// TIA Portal V16 program export: 1 tag tables, 0 data types, 4 data blocks, 6 code blocks (in call order from the OBs), 8 instance data blocks

VAR_GLOBAL   // PLC tag table "Default tag table"
   System_Byte AT %MB1 : Byte;
   FirstScan AT %M1.0 : Bool;
   DiagStatusUpdate AT %M1.1 : Bool;
   AlwaysTRUE AT %M1.2 : Bool;
   AlwaysFALSE AT %M1.3 : Bool;
   Clock_Byte AT %MB0 : Byte;
   Clock_10Hz AT %M0.0 : Bool;
   Clock_5Hz AT %M0.1 : Bool;
   "Clock_2.5Hz" AT %M0.2 : Bool;
   Clock_2Hz AT %M0.3 : Bool;
   "Clock_1.25Hz" AT %M0.4 : Bool;
   Clock_1Hz AT %M0.5 : Bool;
   "Clock_0.625Hz" AT %M0.6 : Bool;
   "Clock_0.5Hz" AT %M0.7 : Bool;
   Aux_1 AT %M2.0 : Bool;
   START_COMM AT %M2.1 : Bool;
   BS_03 AT %M2.6 : Bool;
   Comm_ok AT %M2.3 : Bool;
   Count_Modbus AT %MW50 : Word;
   RST_Count AT %M49.0 : Bool;
   Tag_2 AT %M49.1 : Bool;
   Tag_3 AT %M49.2 : Bool;
   Tag_4 AT %M49.3 : Bool;
   Tag_5 AT %M49.4 : Bool;
   MB_DONE_COUNT AT %MW54 : Word;
   Tag_7 AT %M49.7 : Bool;
   MB_ERROR_COUNT AT %MW58 : Word;
   MB_STATUS AT %MW62 : Word;
   Tag_10 AT %M30.0 : Bool;
   Tag_11 AT %MW70 : Word;
   Tag_12 AT %MW74 : Word;
   Tag_13 AT %MW78 : Word;
   Liga_01 AT %M3.0 : Bool;
   Desliga_01 AT %M3.1 : Bool;
   Liga_02 AT %M3.2 : Bool;
   Desliga_02 AT %M3.3 : Bool;
   Liga_03 AT %M3.4 : Bool;
   Desliga_03 AT %M3.5 : Bool;
   Liga_04 AT %M3.6 : Bool;
   Desliga_04 AT %M3.7 : Bool;
   Liga_05 AT %M4.0 : Bool;
   Desliga_05 AT %M4.1 : Bool;
   Liga_06 AT %M4.2 : Bool;
   Desliga_06 AT %M4.3 : Bool;
   Liga_07 AT %M4.4 : Bool;
   Desliga_07 AT %M4.5 : Bool;
   Liga_08 AT %M4.6 : Bool;
   Desliga_08 AT %M4.7 : Bool;
   Liga_09 AT %M5.0 : Bool;
   Desliga_09 AT %M5.1 : Bool;
   Liga_10 AT %M5.2 : Bool;
   Desliga_10 AT %M5.3 : Bool;
   Liga_11 AT %M5.4 : Bool;
   Desliga_11 AT %M5.5 : Bool;
   Liga_12 AT %M5.6 : Bool;
   Desliga_12 AT %M5.7 : Bool;
   Liga_13 AT %M6.0 : Bool;
   Desliga_13 AT %M6.1 : Bool;
   Liga_14 AT %M6.2 : Bool;
   Desliga_14 AT %M6.3 : Bool;
   Oper_Mode_01 AT %MW80 : Word;
   SP_01 AT %MW82 : Word;
   Oper_Mode_02 AT %MW84 : Word;
   SP_02 AT %MW86 : Word;
   Oper_Mode_03 AT %MW88 : Word;
   SP_03 AT %MW90 : Word;
   Oper_Mode_04 AT %MW92 : Word;
   SP_04 AT %MW94 : Word;
   Oper_Mode_05 AT %MW96 : Word;
   SP_05 AT %MW98 : Word;
   Oper_Mode_06 AT %MW100 : Word;
   SP_06 AT %MW102 : Word;
   Oper_Mode_07 AT %MW104 : Word;
   SP_07 AT %MW106 : Word;
   Oper_Mode_08 AT %MW108 : Word;
   SP_08 AT %MW110 : Word;
   Oper_Mode_09 AT %MW112 : Word;
   SP_09 AT %MW114 : Word;
   Oper_Mode_10 AT %MW116 : Word;
   SP_10 AT %MW118 : Word;
   Oper_Mode_11 AT %MW120 : Word;
   SP_11 AT %MW122 : Word;
   Oper_Mode_12 AT %MW124 : Word;
   SP_12 AT %MW126 : Word;
   Oper_Mode_13 AT %MW128 : Word;
   SP_13 AT %MW130 : Word;
   Oper_Mode_14 AT %MW132 : Word;
   SP_14 AT %MW134 : Word;
   Tag_1 AT %M7.1 : Bool;
   Timeout_Desligado_Counter AT %M6.4 : Bool;
   Timeout_Ligado_Counter AT %M6.5 : Bool;
   Tag_8 AT %M6.6 : Bool;
   Tag_6 AT %M6.7 : Bool;
   MB_CT_DONE AT %M7.2 : Bool;
   MB_CT_ERROR AT %M7.3 : Bool;
   Sts_Auto AT %M7.4 : Bool;
   Tag_9 AT %MW240 : Word;
   Tag_14 AT %MD242 : Real;
   "1" AT %MD246 : Real;
   Tag_15 AT %MW242 : Word;
END_VAR

DATA_BLOCK "Data_block_1"   // DB1
{ S7_Optimized_Access := 'FALSE' }
VERSION : 0.1
// stored: AutoNumber true, DBAccessibleFromOPCUA true, IsOnlyStoredInLoadMemory false, IsWriteProtectedInAS false
   VAR RETAIN
      Descritivo_TBR : Array[0..13] of String;
      Descritivo_TOP : Array[0..1] of String;
   END_VAR
BEGIN
END_DATA_BLOCK

DATA_BLOCK "Modbus"   // DB5
{ S7_Optimized_Access := 'TRUE' }
VERSION : 0.1
// stored: AutoNumber true, DBAccessibleFromOPCUA true, IsOnlyStoredInLoadMemory false, IsRetainMemResEnabled false, IsWriteProtectedInAS false, MemoryReserve 100
   VAR
      Done : Bool;
      Busy : Bool;
      Error : Bool;
      Status : Word;
      Input_Reading : Struct
         "30000" : Array[0..149] of Word;
      END_STRUCT;
   END_VAR
BEGIN
END_DATA_BLOCK

DATA_BLOCK "Modbus_Send_Receive"   // DB10
{ S7_Optimized_Access := 'FALSE' }
VERSION : 0.1
// stored: AutoNumber true, DBAccessibleFromOPCUA true, IsOnlyStoredInLoadMemory false, IsWriteProtectedInAS false
   VAR
      "30001" : Word;
      "30002" : Word;   // COMM_OK = 3FFF
      "32001" : Word;   // STS_UNIT_01
      "32002" : Word;   // OPER_UNIT_01
      "32003" : Word;   // SP_UNIT_01
      "32004" : Word;   // ERROR_UNIT_01
      "32005" : Word;   // PV_UNIT_01
      "32006" : Word;   // SERROR_UNIT_01
      "32007" : Word;   // STS_UNIT_02
      "32008" : Word;   // OPER_UNIT_02
      "32009" : Word;   // SP_UNIT_02
      "32010" : Word;   // ERROR_UNIT_02
      "32011" : Word;   // PV_UNIT_02
      "32012" : Word;   // SERROR_UNIT_02
      "32013" : Word;
      "32014" : Word;
      "32015" : Word;
      "32016" : Word;
      "32017" : Word;
      "32018" : Word;
      "32019" : Word;
      "32020" : Word;
      "32021" : Word;
      "32022" : Word;
      "32023" : Word;
      "32024" : Word;
      "32025" : Word;
      "32026" : Word;
      "32027" : Word;
      "32028" : Word;
      "32029" : Word;
      "32030" : Word;
      "32031" : Word;
      "32032" : Word;
      "32033" : Word;
      "32034" : Word;
      "32035" : Word;
      "32036" : Word;
      "32037" : Word;
      "32038" : Word;
      "32039" : Word;
      "32040" : Word;
      "32041" : Word;
      "32042" : Word;
      "32043" : Word;
      "32044" : Word;
      "32045" : Word;
      "32046" : Word;
      "32047" : Word;
      "32048" : Word;
      "32049" : Word;
      "32050" : Word;
      "32051" : Word;
      "32052" : Word;
      "32053" : Word;
      "32054" : Word;
      "32055" : Word;
      "32056" : Word;
      "32057" : Word;
      "32058" : Word;
      "32059" : Word;
      "32060" : Word;
      "32061" : Word;
      "32062" : Word;
      "32063" : Word;
      "32064" : Word;
      "32065" : Word;
      "32066" : Word;
      "32067" : Word;
      "32068" : Word;
      "32069" : Word;
      "32070" : Word;
      "32071" : Word;
      "32072" : Word;
      "32073" : Word;
      "32074" : Word;
      "32075" : Word;
      "32076" : Word;
      "32077" : Word;
      "32078" : Word;
      "32079" : Word;
      "32080" : Word;
      "32081" : Word;
      "32082" : Word;
      "32083" : Word;
      "32084" : Word;
      "40001" : Word;   // COMM
      "42001" : Word;   // STS
      "42002" : Word;   // OPER_MODE
      "42003" : Word;   // SP
      "42004" : Word;   // STS
      "42005" : Word;   // OPER_MODE
      "42006" : Word;   // SP
      "42007" : Word;   // STS
      "42008" : Word;   // OPER_MODE
      "42009" : Word;   // SP
      "42010" : Word;   // STS
      "42011" : Word;   // OPER_MODE
      "42012" : Word;   // SP
      "42013" : Word;   // STS
      "42014" : Word;   // OPER_MODE
      "42015" : Word;   // SP
      "42016" : Word;   // STS
      "42017" : Word;   // OPER_MODE
      "42018" : Word;   // SP
      "42019" : Word;   // STS
      "42020" : Word;   // OPER_MODE
      "42021" : Word;   // SP
      "42022" : Word;   // STS
      "42023" : Word;   // OPER_MODE
      "42024" : Word;   // SP
      "42025" : Word;   // STS
      "42026" : Word;   // OPER_MODE
      "42027" : Word;   // SP
      "42028" : Word;   // STS
      "42029" : Word;   // OPER_MODE
      "42030" : Word;   // SP
      "42031" : Word;   // STS
      "42032" : Word;   // OPER_MODE
      "42033" : Word;   // SP
      "42034" : Word;   // STS
      "42035" : Word;   // OPER_MODE
      "42036" : Word;   // SP
      "42037" : Word;   // STS
      "42038" : Word;   // OPER_MODE
      "42039" : Word;   // SP
      "42040" : Word;   // STS
      "42041" : Word;   // OPER_MODE
      "42042" : Word;   // SP
      Extrusora_1 : Struct
         Ligado : Bool;
         Fan : Bool;
         Heating : Bool;
         Cooling : Bool;
         Sts_Fan : Bool;
         Sts_Heating : Bool;
         Sts_Cooling : Bool;
         Slave : Bool;
         Master : Bool;
         SP : Real;
         PV : Real;
      END_STRUCT;
      Extrusora_2 : Struct
         Ligado : Bool;
         Fan : Bool;
         Heating : Bool;
         Cooling : Bool;
         Sts_Fan : Bool;
         Sts_Heating : Bool;
         Sts_Cooling : Bool;
         Slave : Bool;
         Master : Bool;
         SP : Real;
         PV : Real;
      END_STRUCT;
      Extrusora_3 : Struct
         Ligado : Bool;
         Fan : Bool;
         Heating : Bool;
         Cooling : Bool;
         Sts_Fan : Bool;
         Sts_Heating : Bool;
         Sts_Cooling : Bool;
         Slave : Bool;
         Master : Bool;
         SP : Real;
         PV : Real;
      END_STRUCT;
      Extrusora_4 : Struct
         Ligado : Bool;
         Fan : Bool;
         Heating : Bool;
         Cooling : Bool;
         Sts_Fan : Bool;
         Sts_Heating : Bool;
         Sts_Cooling : Bool;
         Slave : Bool;
         Master : Bool;
         SP : Real;
         PV : Real;
      END_STRUCT;
      Extrusora_5 : Struct
         Ligado : Bool;
         Fan : Bool;
         Heating : Bool;
         Cooling : Bool;
         Sts_Fan : Bool;
         Sts_Heating : Bool;
         Sts_Cooling : Bool;
         Slave : Bool;
         Master : Bool;
         SP : Real;
         PV : Real;
      END_STRUCT;
      Extrusora_6 : Struct
         Ligado : Bool;
         Fan : Bool;
         Heating : Bool;
         Cooling : Bool;
         Sts_Fan : Bool;
         Sts_Heating : Bool;
         Sts_Cooling : Bool;
         Slave : Bool;
         Master : Bool;
         SP : Real;
         PV : Real;
      END_STRUCT;
      Extrusora_7 : Struct
         Ligado : Bool;
         Fan : Bool;
         Heating : Bool;
         Cooling : Bool;
         Sts_Fan : Bool;
         Sts_Heating : Bool;
         Sts_Cooling : Bool;
         Slave : Bool;
         Master : Bool;
         SP : Real;
         PV : Real;
      END_STRUCT;
      Extrusora_8 : Struct
         Ligado : Bool;
         Fan : Bool;
         Heating : Bool;
         Cooling : Bool;
         Sts_Fan : Bool;
         Sts_Heating : Bool;
         Sts_Cooling : Bool;
         Slave : Bool;
         Master : Bool;
         SP : Real;
         PV : Real;
      END_STRUCT;
      Extrusora_9 : Struct
         Ligado : Bool;
         Fan : Bool;
         Heating : Bool;
         Cooling : Bool;
         Sts_Fan : Bool;
         Sts_Heating : Bool;
         Sts_Cooling : Bool;
         Slave : Bool;
         Master : Bool;
         SP : Real;
         PV : Real;
      END_STRUCT;
      Extrusora_10 : Struct
         Ligado : Bool;
         Fan : Bool;
         Heating : Bool;
         Cooling : Bool;
         Sts_Fan : Bool;
         Sts_Heating : Bool;
         Sts_Cooling : Bool;
         Slave : Bool;
         Master : Bool;
         SP : Real;
         PV : Real;
      END_STRUCT;
      Extrusora_11 : Struct
         Ligado : Bool;
         Fan : Bool;
         Heating : Bool;
         Cooling : Bool;
         Sts_Fan : Bool;
         Sts_Heating : Bool;
         Sts_Cooling : Bool;
         Slave : Bool;
         Master : Bool;
         SP : Real;
         PV : Real;
      END_STRUCT;
      Extrusora_12 : Struct
         Ligado : Bool;
         Fan : Bool;
         Heating : Bool;
         Cooling : Bool;
         Sts_Fan : Bool;
         Sts_Heating : Bool;
         Sts_Cooling : Bool;
         Slave : Bool;
         Master : Bool;
         SP : Real;
         PV : Real;
      END_STRUCT;
      Extrusora_13 : Struct
         Ligado : Bool;
         Fan : Bool;
         Heating : Bool;
         Cooling : Bool;
         Sts_Fan : Bool;
         Sts_Heating : Bool;
         Sts_Cooling : Bool;
         Slave : Bool;
         Master : Bool;
         SP : Real;
         PV : Real;
      END_STRUCT;
      Extrusora_14 : Struct
         Ligado : Bool;
         Fan : Bool;
         Heating : Bool;
         Cooling : Bool;
         Sts_Fan : Bool;
         Sts_Heating : Bool;
         Sts_Cooling : Bool;
         Slave : Bool;
         Master : Bool;
         SP : Real;
         PV : Real;
      END_STRUCT;
      Malfunction_1 : Bool;
      Malfunction_2 : Bool;
      Malfunction_3 : Bool;
      Malfunction_4 : Bool;
      Malfunction_5 : Bool;
      Malfunction_6 : Bool;
      Malfunction_7 : Bool;
      Malfunction_8 : Bool;
      Malfunction_9 : Bool;
      Malfunction_10 : Bool;
      Malfunction_11 : Bool;
      Malfunction_12 : Bool;
      Malfunction_13 : Bool;
      Malfunction_14 : Bool;
   END_VAR
BEGIN
END_DATA_BLOCK

DATA_BLOCK "Modbus_Send_Receive_1"   // DB13
{ S7_Optimized_Access := 'FALSE' }
VERSION : 0.1
// stored: AutoNumber false, DBAccessibleFromOPCUA true, IsOnlyStoredInLoadMemory false, IsWriteProtectedInAS false
   VAR
      Reading_Struct : Struct
         "32001" : Word;   // STS_UNIT_01
         "32002" : Word;   // OPER_UNIT_01
         "32003" : Word;   // SP_UNIT_01
         "32004" : Word;   // ERROR_UNIT_01
         "32005" : Word;   // PV_UNIT_01
         "32006" : Word;   // SERROR_UNIT_01
         "32007" : Word;   // STS_UNIT_02
         "32008" : Word;   // OPER_UNIT_02
         "32009" : Word;   // SP_UNIT_02
         "32010" : Word;   // ERROR_UNIT_02
         "32011" : Word;   // PV_UNIT_02
         "32012" : Word;   // SERROR_UNIT_02
         "32013" : Word;   // STS_UNIT_01
         "32014" : Word;   // OPER_UNIT_01
         "32015" : Word;   // SP_UNIT_01
         "32016" : Word;   // ERROR_UNIT_01
         "32017" : Word;   // PV_UNIT_01
         "32018" : Word;   // SERROR_UNIT_01
         "32019" : Word;   // STS_UNIT_02
         "32020" : Word;   // OPER_UNIT_02
         "32021" : Word;   // SP_UNIT_02
         "32022" : Word;   // ERROR_UNIT_02
         "32023" : Word;   // PV_UNIT_02
         "32024" : Word;   // SERROR_UNIT_02
         "32025" : Word;   // STS_UNIT_01
         "32026" : Word;   // OPER_UNIT_01
         "32027" : Word;   // SP_UNIT_01
         "32028" : Word;   // ERROR_UNIT_01
         "32029" : Word;   // PV_UNIT_01
         "32030" : Word;   // SERROR_UNIT_01
         "32031" : Word;   // STS_UNIT_02
         "32032" : Word;   // OPER_UNIT_02
         "32033" : Word;   // SP_UNIT_02
         "32034" : Word;   // ERROR_UNIT_02
         "32035" : Word;   // PV_UNIT_02
         "32036" : Word;   // SERROR_UNIT_02
         "32037" : Word;   // STS_UNIT_01
         "32038" : Word;   // OPER_UNIT_01
         "32039" : Word;   // SP_UNIT_01
         "32040" : Word;   // ERROR_UNIT_01
         "32041" : Word;   // PV_UNIT_01
         "32042" : Word;   // SERROR_UNIT_01
         "32043" : Word;   // STS_UNIT_02
         "32044" : Word;   // OPER_UNIT_02
         "32045" : Word;   // SP_UNIT_02
         "32046" : Word;   // ERROR_UNIT_02
         "32047" : Word;   // PV_UNIT_02
         "32048" : Word;   // SERROR_UNIT_02
         "32049" : Word;   // STS_UNIT_01
         "32050" : Word;   // OPER_UNIT_01
         "32051" : Word;   // SP_UNIT_01
         "32052" : Word;   // ERROR_UNIT_01
         "32053" : Word;   // PV_UNIT_01
         "32054" : Word;   // SERROR_UNIT_01
         "32055" : Word;   // STS_UNIT_02
         "32056" : Word;   // OPER_UNIT_02
         "32057" : Word;   // SP_UNIT_02
         "32058" : Word;   // ERROR_UNIT_02
         "32059" : Word;   // PV_UNIT_02
         "32060" : Word;   // SERROR_UNIT_02
         "32061" : Word;   // STS_UNIT_01
         "32062" : Word;   // OPER_UNIT_01
         "32063" : Word;   // SP_UNIT_01
         "32064" : Word;   // ERROR_UNIT_01
         "32065" : Word;   // PV_UNIT_01
         "32066" : Word;   // SERROR_UNIT_01
         "32067" : Word;   // STS_UNIT_02
         "32068" : Word;   // OPER_UNIT_02
         "32069" : Word;   // SP_UNIT_02
         "32070" : Word;   // ERROR_UNIT_02
         "32071" : Word;   // PV_UNIT_02
         "32072" : Word;   // SERROR_UNIT_02
         "32073" : Word;   // STS_UNIT_01
         "32074" : Word;   // OPER_UNIT_01
         "32075" : Word;   // SP_UNIT_01
         "32076" : Word;   // ERROR_UNIT_01
         "32077" : Word;   // PV_UNIT_01
         "32078" : Word;   // SERROR_UNIT_01
         "32079" : Word;   // STS_UNIT_02
         "32080" : Word;   // OPER_UNIT_02
         "32081" : Word;   // SP_UNIT_02
         "32082" : Word;   // ERROR_UNIT_02
         "32083" : Word;   // PV_UNIT_02
         "32084" : Word;   // SERROR_UNIT_02
         "40001" : Word;
         "42001" : Word;   // STS
         "42002" : Word;   // OPER_MODE
         "42003" : Word;   // SP
         "42004" : Word;
         "42005" : Word;
         "42006" : Word;
         "42007" : Word;
         "42008" : Word;
         "42009" : Word;
         "42010" : Word;
         "42011" : Word;
         "42012" : Word;
         "42013" : Word;
         "42014" : Word;
         "42015" : Word;
         "42016" : Word;
         "42017" : Word;
         "42018" : Word;
         "42019" : Word;
         "42020" : Word;
         "42021" : Word;
         "42022" : Word;
         "42023" : Word;
         "42024" : Word;
         "42025" : Word;
         "42026" : Word;
         "42027" : Word;
         "42028" : Word;
         "42029" : Word;
         "42030" : Word;
         "42031" : Word;
         "42032" : Word;
         "42033" : Word;
         "42034" : Word;
         "42035" : Word;
         "42036" : Word;
         "42037" : Word;
         "42038" : Word;
         "42039" : Word;
         "42040" : Word;
         "42041" : Word;
         "42042" : Word;
      END_STRUCT;
      Reading_Struct_2 : Struct
         "30001" : Word;
         "30002" : Word;   // COMM_OK = 3FFF
      END_STRUCT;
      Extrusora_1 : Struct
         Ligado : Bool;
         Fan : Bool;
         Heating : Bool;
         Cooling : Bool;
         Sts_Fan : Bool;
         Sts_Heating : Bool;
         Sts_Cooling : Bool;
         Slave : Bool;
         Master : Bool;
         SP : Word;
         PV : Word;
      END_STRUCT;
      Extrusora_2 : Struct
         Ligado : Bool;
         Fan : Bool;
         Heating : Bool;
         Cooling : Bool;
         Sts_Fan : Bool;
         Sts_Heating : Bool;
         Sts_Cooling : Bool;
         Slave : Bool;
         Master : Bool;
         SP : Word;
         PV : Word;
      END_STRUCT;
      Extrusora_3 : Struct
         Ligado : Bool;
         Fan : Bool;
         Heating : Bool;
         Cooling : Bool;
         Sts_Fan : Bool;
         Sts_Heating : Bool;
         Sts_Cooling : Bool;
         Slave : Bool;
         Master : Bool;
         SP : Word;
         PV : Word;
      END_STRUCT;
      Extrusora_4 : Struct
         Ligado : Bool;
         Fan : Bool;
         Heating : Bool;
         Cooling : Bool;
         Sts_Fan : Bool;
         Sts_Heating : Bool;
         Sts_Cooling : Bool;
         Slave : Bool;
         Master : Bool;
         SP : Word;
         PV : Word;
      END_STRUCT;
      Extrusora_5 : Struct
         Ligado : Bool;
         Fan : Bool;
         Heating : Bool;
         Cooling : Bool;
         Sts_Fan : Bool;
         Sts_Heating : Bool;
         Sts_Cooling : Bool;
         Slave : Bool;
         Master : Bool;
         SP : Word;
         PV : Word;
      END_STRUCT;
      Extrusora_6 : Struct
         Ligado : Bool;
         Fan : Bool;
         Heating : Bool;
         Cooling : Bool;
         Sts_Fan : Bool;
         Sts_Heating : Bool;
         Sts_Cooling : Bool;
         Slave : Bool;
         Master : Bool;
         SP : Word;
         PV : Word;
      END_STRUCT;
      Extrusora_7 : Struct
         Ligado : Bool;
         Fan : Bool;
         Heating : Bool;
         Cooling : Bool;
         Sts_Fan : Bool;
         Sts_Heating : Bool;
         Sts_Cooling : Bool;
         Slave : Bool;
         Master : Bool;
         SP : Word;
         PV : Word;
      END_STRUCT;
      Extrusora_8 : Struct
         Ligado : Bool;
         Fan : Bool;
         Heating : Bool;
         Cooling : Bool;
         Sts_Fan : Bool;
         Sts_Heating : Bool;
         Sts_Cooling : Bool;
         Slave : Bool;
         Master : Bool;
         SP : Word;
         PV : Word;
      END_STRUCT;
      Extrusora_9 : Struct
         Ligado : Bool;
         Fan : Bool;
         Heating : Bool;
         Cooling : Bool;
         Sts_Fan : Bool;
         Sts_Heating : Bool;
         Sts_Cooling : Bool;
         Slave : Bool;
         Master : Bool;
         SP : Word;
         PV : Word;
      END_STRUCT;
      Extrusora_10 : Struct
         Ligado : Bool;
         Fan : Bool;
         Heating : Bool;
         Cooling : Bool;
         Sts_Fan : Bool;
         Sts_Heating : Bool;
         Sts_Cooling : Bool;
         Slave : Bool;
         Master : Bool;
         SP : Word;
         PV : Word;
      END_STRUCT;
      Extrusora_11 : Struct
         Ligado : Bool;
         Fan : Bool;
         Heating : Bool;
         Cooling : Bool;
         Sts_Fan : Bool;
         Sts_Heating : Bool;
         Sts_Cooling : Bool;
         Slave : Bool;
         Master : Bool;
         SP : Word;
         PV : Word;
      END_STRUCT;
      Extrusora_12 : Struct
         Ligado : Bool;
         Fan : Bool;
         Heating : Bool;
         Cooling : Bool;
         Sts_Fan : Bool;
         Sts_Heating : Bool;
         Sts_Cooling : Bool;
         Slave : Bool;
         Master : Bool;
         SP : Word;
         PV : Word;
      END_STRUCT;
      Extrusora_13 : Struct
         Ligado : Bool;
         Fan : Bool;
         Heating : Bool;
         Cooling : Bool;
         Sts_Fan : Bool;
         Sts_Heating : Bool;
         Sts_Cooling : Bool;
         Slave : Bool;
         Master : Bool;
         SP : Word;
         PV : Word;
      END_STRUCT;
      Extrusora_14 : Struct
         Ligado : Bool;
         Fan : Bool;
         Heating : Bool;
         Cooling : Bool;
         Sts_Fan : Bool;
         Sts_Heating : Bool;
         Sts_Cooling : Bool;
         Slave : Bool;
         Master : Bool;
         SP : Word;
         PV : Word;
      END_STRUCT;
      Malfunction_1 : Bool;
      Malfunction_2 : Bool;
      Malfunction_3 : Bool;
      Malfunction_4 : Bool;
      Malfunction_5 : Bool;
      Malfunction_6 : Bool;
      Malfunction_7 : Bool;
      Malfunction_8 : Bool;
      Malfunction_9 : Bool;
      Malfunction_10 : Bool;
      Malfunction_11 : Bool;
      Malfunction_12 : Bool;
      Malfunction_13 : Bool;
      Malfunction_14 : Bool;
   END_VAR
BEGIN
END_DATA_BLOCK

ORGANIZATION_BLOCK "Main"   // OB1, LAD, ProgramCycle
TITLE = "Main Program Sweep (Cycle)"
{ S7_Optimized_Access := 'TRUE' }
VERSION : 0.1
// stored: AutoNumber true, IsIECCheckEnabled false, SetENOAutomatically false
BEGIN

REGION Network 1: Start modbus comm
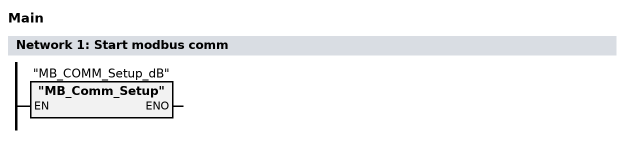
   RUNG wire#powerrail
      "MB_COMM_Setup_dB"()
   END_RUNG
   // the same network as SCL:
   "MB_COMM_Setup_dB"();   // "MB_Comm_Setup"
END_REGION
END_ORGANIZATION_BLOCK

FUNCTION_BLOCK "MB_Comm_Setup"   // FB1, LAD
{ S7_Optimized_Access := 'FALSE' }
VERSION : 0.1
// stored: AutoNumber true, IsIECCheckEnabled false, SetENOAutomatically false, UDAEnableTagReadback false
   VAR DB_SPECIFIC
      Input_Registers_3000X_In { ExternalAccessible := 'False'; ExternalVisible := 'False'; ExternalWritable := 'False'} : Struct
         "3000X" { ExternalAccessible := 'False'; ExternalVisible := 'False'; ExternalWritable := 'False'} : Array[0..150] of Word;
      END_STRUCT;
   END_VAR
   VAR
      Input_Registers_In_AT AT Input_Registers_3000X_In : Struct
         "30001" : Array[0..15] of Bool;
         "30001_2" : Array[0..15] of Bool;   // Status of the Adaptor
         "30002" : Array[0..15] of Bool;   // Indoor Unit Connection Status
         "30003" : Array[0..15] of Bool;   // Empty
         "30004" : Array[0..15] of Bool;   // Empty
         "30005" : Array[0..15] of Bool;   // Empty
         "30006" : Array[0..15] of Bool;   // Indoor Unit Communication Status
         "31001" : Array[0..15] of Bool;   // Various
         "31002" : Array[0..15] of Bool;   // 1st word - Indoor unit cooling setpoint upper limit, 2 - word indoor unit cooling setpoint lower limit
         "31003" : Array[0..15] of Bool;   // 1st word - Indoor unit heating setpoint upper limit, 2 - word indoor unit heating setpoint lower limit
         "31004" : Array[0..15] of Bool;   // Various
         "31005" : Array[0..15] of Bool;   // 1st word - Indoor unit cooling setpoint upper limit, 2 - word indoor unit cooling setpoint lower limit
         "31006" : Array[0..15] of Bool;   // 1st word - Indoor unit heating setpoint upper limit, 2 - word indoor unit heating setpoint lower limit
         "31007" : Array[0..15] of Bool;   // Various
         "31008" : Array[0..15] of Bool;   // 1st word - Indoor unit cooling setpoint upper limit, 2 - word indoor unit cooling setpoint lower limit
         "31009" : Array[0..15] of Bool;   // 1st word - Indoor unit heating setpoint upper limit, 2 - word indoor unit heating setpoint lower limit
         "31010" : Array[0..15] of Bool;   // Various
         "31011" : Array[0..15] of Bool;   // 1st word - Indoor unit cooling setpoint upper limit, 2 - word indoor unit cooling setpoint lower limit
         "31012" : Array[0..15] of Bool;   // 1st word - Indoor unit heating setpoint upper limit, 2 - word indoor unit heating setpoint lower limit
         "31013" : Array[0..15] of Bool;   // Various
         "31014" : Array[0..15] of Bool;   // 1st word - Indoor unit cooling setpoint upper limit, 2 - word indoor unit cooling setpoint lower limit
         "31015" : Array[0..15] of Bool;   // 1st word - Indoor unit heating setpoint upper limit, 2 - word indoor unit heating setpoint lower limit
         "31016" : Array[0..15] of Bool;   // Various
         "31017" : Array[0..15] of Bool;   // 1st word - Indoor unit cooling setpoint upper limit, 2 - word indoor unit cooling setpoint lower limit
         "31018" : Array[0..15] of Bool;   // 1st word - Indoor unit heating setpoint upper limit, 2 - word indoor unit heating setpoint lower limit
         "31019" : Array[0..15] of Bool;   // Various
         "31020" : Array[0..15] of Bool;   // 1st word - Indoor unit cooling setpoint upper limit, 2 - word indoor unit cooling setpoint lower limit
         "31021" : Array[0..15] of Bool;   // 1st word - Indoor unit heating setpoint upper limit, 2 - word indoor unit heating setpoint lower limit
         "31022" : Array[0..15] of Bool;   // Various
         "31023" : Array[0..15] of Bool;   // 1st word - Indoor unit cooling setpoint upper limit, 2 - word indoor unit cooling setpoint lower limit
         "31024" : Array[0..15] of Bool;   // 1st word - Indoor unit heating setpoint upper limit, 2 - word indoor unit heating setpoint lower limit
         "31025" : Array[0..15] of Bool;   // Various
         "31026" : Array[0..15] of Bool;   // 1st word - Indoor unit cooling setpoint upper limit, 2 - word indoor unit cooling setpoint lower limit
         "31027" : Array[0..15] of Bool;   // 1st word - Indoor unit heating setpoint upper limit, 2 - word indoor unit heating setpoint lower limit
         "31028" : Array[0..15] of Bool;   // Various
         "31029" : Array[0..15] of Bool;   // 1st word - Indoor unit cooling setpoint upper limit, 2 - word indoor unit cooling setpoint lower limit
         "31030" : Array[0..15] of Bool;   // 1st word - Indoor unit heating setpoint upper limit, 2 - word indoor unit heating setpoint lower limit
         "31031" : Array[0..15] of Bool;   // Various
         "31032" : Array[0..15] of Bool;   // 1st word - Indoor unit cooling setpoint upper limit, 2 - word indoor unit cooling setpoint lower limit
         "31033" : Array[0..15] of Bool;   // 1st word - Indoor unit heating setpoint upper limit, 2 - word indoor unit heating setpoint lower limit
         "31034" : Array[0..15] of Bool;   // Various
         "31035" : Array[0..15] of Bool;   // 1st word - Indoor unit cooling setpoint upper limit, 2 - word indoor unit cooling setpoint lower limit
         "31036" : Array[0..15] of Bool;   // 1st word - Indoor unit heating setpoint upper limit, 2 - word indoor unit heating setpoint lower limit
         "31037" : Array[0..15] of Bool;   // Various
         "31038" : Array[0..15] of Bool;   // 1st word - Indoor unit cooling setpoint upper limit, 2 - word indoor unit cooling setpoint lower limit
         "31039" : Array[0..15] of Bool;   // 1st word - Indoor unit heating setpoint upper limit, 2 - word indoor unit heating setpoint lower limit
         "31040" : Array[0..15] of Bool;   // Various
         "31041" : Array[0..15] of Bool;   // 1st word - Indoor unit cooling setpoint upper limit, 2 - word indoor unit cooling setpoint lower limit
         "31042" : Array[0..15] of Bool;   // 1st word - Indoor unit heating setpoint upper limit, 2 - word indoor unit heating setpoint lower limit
         "31043" : Array[0..15] of Bool;   // Various
         "31044" : Array[0..15] of Bool;   // 1st word - Indoor unit cooling setpoint upper limit, 2 - word indoor unit cooling setpoint lower limit
         "31045" : Array[0..15] of Bool;   // 1st word - Indoor unit heating setpoint upper limit, 2 - word indoor unit heating setpoint lower limit
         "31046" : Array[0..15] of Bool;   // Various
         "31047" : Array[0..15] of Bool;   // 1st word - Indoor unit cooling setpoint upper limit, 2 - word indoor unit cooling setpoint lower limit
         "31048" : Array[0..15] of Bool;   // 1st word - Indoor unit heating setpoint upper limit, 2 - word indoor unit heating setpoint lower limit
         "32001" : Array[0..15] of Bool;   // Important stuff
         "32002" : Array[0..15] of Bool;   // Important stuff_2
         "32003" : Array[0..15] of Bool;   // Setpoint Temperature
         "32004" : Array[0..15] of Bool;   // Important Stuff_3
         "32005" : Array[0..15] of Bool;   // Room Temperature
         "32006" : Array[0..15] of Bool;   // Error
         "32007" : Array[0..15] of Bool;   // Important stuff
         "32008" : Array[0..15] of Bool;   // Important stuff_2
         "32009" : Array[0..15] of Bool;   // Setpoint Temperature
         "32010" : Array[0..15] of Bool;   // Important Stuff_3
         "32011" : Array[0..15] of Bool;   // Room Temperature
         "32012" : Array[0..15] of Bool;   // Error
         "32013" : Array[0..15] of Bool;   // Important stuff
         "32014" : Array[0..15] of Bool;   // Important stuff_2
         "32015" : Array[0..15] of Bool;   // Setpoint Temperature
         "32016" : Array[0..15] of Bool;   // Important Stuff_3
         "32017" : Array[0..15] of Bool;   // Room Temperature
         "32018" : Array[0..15] of Bool;   // Error
         "32019" : Array[0..15] of Bool;   // Important stuff
         "32020" : Array[0..15] of Bool;   // Important stuff_2
         "32021" : Array[0..15] of Bool;   // Setpoint Temperature
         "32022" : Array[0..15] of Bool;   // Important Stuff_3
         "32023" : Array[0..15] of Bool;   // Room Temperature
         "32024" : Array[0..15] of Bool;   // Error
         "32025" : Array[0..15] of Bool;   // Important stuff
         "32026" : Array[0..15] of Bool;   // Important stuff_2
         "32027" : Array[0..15] of Bool;   // Setpoint Temperature
         "32028" : Array[0..15] of Bool;   // Important Stuff_3
         "32029" : Array[0..15] of Bool;   // Room Temperature
         "32030" : Array[0..15] of Bool;   // Error
         "32031" : Array[0..15] of Bool;   // Important stuff
         "32032" : Array[0..15] of Bool;   // Important stuff_2
         "32033" : Array[0..15] of Bool;   // Setpoint Temperature
         "32034" : Array[0..15] of Bool;   // Important Stuff_3
         "32035" : Array[0..15] of Bool;   // Room Temperature
         "32036" : Array[0..15] of Bool;   // Error
         "32037" : Array[0..15] of Bool;   // Important stuff
         "32038" : Array[0..15] of Bool;   // Important stuff_2
         "32039" : Array[0..15] of Bool;   // Setpoint Temperature
         "32040" : Array[0..15] of Bool;   // Important Stuff_3
         "32041" : Array[0..15] of Bool;   // Room Temperature
         "32042" : Array[0..15] of Bool;   // Error
         "32043" : Array[0..15] of Bool;   // Important stuff
         "32044" : Array[0..15] of Bool;   // Important stuff_2
         "32045" : Array[0..15] of Bool;   // Setpoint Temperature
         "32046" : Array[0..15] of Bool;   // Important Stuff_3
         "32047" : Array[0..15] of Bool;   // Room Temperature
         "32048" : Array[0..15] of Bool;   // Error
         "32049" : Array[0..15] of Bool;   // Important stuff
         "32050" : Array[0..15] of Bool;   // Important stuff_2
         "32051" : Array[0..15] of Bool;   // Setpoint Temperature
         "32052" : Array[0..15] of Bool;   // Important Stuff_3
         "32053" : Array[0..15] of Bool;   // Room Temperature
         "32054" : Array[0..15] of Bool;   // Error
         "32055" : Array[0..15] of Bool;   // Important stuff
         "32056" : Array[0..15] of Bool;   // Important stuff_2
         "32057" : Array[0..15] of Bool;   // Setpoint Temperature
         "32058" : Array[0..15] of Bool;   // Important Stuff_3
         "32059" : Array[0..15] of Bool;   // Room Temperature
         "32060" : Array[0..15] of Bool;   // Error
         "32061" : Array[0..15] of Bool;   // Important stuff
         "32062" : Array[0..15] of Bool;   // Important stuff_2
         "32063" : Array[0..15] of Bool;   // Setpoint Temperature
         "32064" : Array[0..15] of Bool;   // Important Stuff_3
         "32065" : Array[0..15] of Bool;   // Room Temperature
         "32066" : Array[0..15] of Bool;   // Error
         "32067" : Array[0..15] of Bool;   // Important stuff
         "32068" : Array[0..15] of Bool;   // Important stuff_2
         "32069" : Array[0..15] of Bool;   // Setpoint Temperature
         "32070" : Array[0..15] of Bool;   // Important Stuff_3
         "32071" : Array[0..15] of Bool;   // Room Temperature
         "32072" : Array[0..15] of Bool;   // Error
         "32073" : Array[0..15] of Bool;   // Important stuff
         "32074" : Array[0..15] of Bool;   // Important stuff_2
         "32075" : Array[0..15] of Bool;   // Setpoint Temperature
         "32076" : Array[0..15] of Bool;   // Important Stuff_3
         "32077" : Array[0..15] of Bool;   // Room Temperature
         "32078" : Array[0..15] of Bool;   // Error
         "32079" : Array[0..15] of Bool;   // Important stuff
         "32080" : Array[0..15] of Bool;   // Important stuff_2
         "32081" : Array[0..15] of Bool;   // Setpoint Temperature
         "32082" : Array[0..15] of Bool;   // Important Stuff_3
         "32083" : Array[0..15] of Bool;   // Room Temperature
         "32084" : Array[0..15] of Bool;   // Error
         "32085" : Array[0..15] of Bool;   // Important stuff
         "32086" : Array[0..15] of Bool;   // Important stuff_2
         "32087" : Array[0..15] of Bool;   // Setpoint Temperature
         "32088" : Array[0..15] of Bool;   // Important Stuff_3
         "32089" : Array[0..15] of Bool;   // Room Temperature
         "32090" : Array[0..15] of Bool;   // Error
         "32091" : Array[0..15] of Bool;   // Important stuff
         "32092" : Array[0..15] of Bool;   // Important stuff_2
         "32093" : Array[0..15] of Bool;   // Setpoint Temperature
         "32094" : Array[0..15] of Bool;   // Important Stuff_3
         "32095" : Array[0..15] of Bool;   // Room Temperature
         "32096" : Array[0..15] of Bool;   // Error
      END_STRUCT;
   END_VAR
   // // Input_Registers_3000X_In."3000X"[0] : 30001
   // // Input_Registers_In_AT."30004"[0] : Fan Mode Capability
   // // Input_Registers_In_AT."30004"[1] : Cooling Mode Capability
   // // Input_Registers_In_AT."30004"[2] : Heating Mode Capability
   // // Input_Registers_In_AT."30004"[3] : Auto Mode Capability
   // // Input_Registers_In_AT."30004"[4] : Dry Mode Capability
   // // Input_Registers_In_AT."30004"[8] : Fan Direction Level Capability
   // // Input_Registers_In_AT."30004"[9] : Fan Direction Level Capability
   // // Input_Registers_In_AT."30004"[10] : Fan Direction Level Capability
   // // Input_Registers_In_AT."30004"[11] : Fan Direction Capability
   // // Input_Registers_In_AT."30004"[12] : Fan Volume Level Capability
   // // Input_Registers_In_AT."30004"[13] : Fan Volume Level Capability
   // // Input_Registers_In_AT."30004"[14] : Fan Volume Level Capability
   // // Input_Registers_In_AT."30004"[15] : Fan Volume Capability
   // // Input_Registers_In_AT."30005"[0] : Fan Mode Capability
   // // Input_Registers_In_AT."30005"[1] : Cooling Mode Capability
   // // Input_Registers_In_AT."30005"[2] : Heating Mode Capability
   // // Input_Registers_In_AT."30005"[3] : Auto Mode Capability
   // // Input_Registers_In_AT."30005"[4] : Dry Mode Capability
   // // Input_Registers_In_AT."30005"[8] : Fan Direction Level Capability
   // // Input_Registers_In_AT."30005"[9] : Fan Direction Level Capability
   // // Input_Registers_In_AT."30005"[10] : Fan Direction Level Capability
   // // Input_Registers_In_AT."30005"[11] : Fan Direction Capability
   // // Input_Registers_In_AT."30005"[12] : Fan Volume Level Capability
   // // Input_Registers_In_AT."30005"[13] : Fan Volume Level Capability
   // // Input_Registers_In_AT."30005"[14] : Fan Volume Level Capability
   // // Input_Registers_In_AT."30005"[15] : Fan Volume Capability
   // // Input_Registers_In_AT."31001"[0] : Fan Mode Capability
   // // Input_Registers_In_AT."31001"[1] : Cooling Mode Capability
   // // Input_Registers_In_AT."31001"[2] : Heating Mode Capability
   // // Input_Registers_In_AT."31001"[3] : Auto Mode Capability
   // // Input_Registers_In_AT."31001"[4] : Dry Mode Capability
   // // Input_Registers_In_AT."31001"[8] : Fan Direction Level Capability
   // // Input_Registers_In_AT."31001"[9] : Fan Direction Level Capability
   // // Input_Registers_In_AT."31001"[10] : Fan Direction Level Capability
   // // Input_Registers_In_AT."31001"[11] : Fan Direction Capability
   // // Input_Registers_In_AT."31001"[12] : Fan Volume Level Capability
   // // Input_Registers_In_AT."31001"[13] : Fan Volume Level Capability
   // // Input_Registers_In_AT."31001"[14] : Fan Volume Level Capability
   // // Input_Registers_In_AT."31001"[15] : Fan Volume Capability
   // // Input_Registers_In_AT."31004"[0] : Fan Mode Capability
   // // Input_Registers_In_AT."31004"[1] : Cooling Mode Capability
   // // Input_Registers_In_AT."31004"[2] : Heating Mode Capability
   // // Input_Registers_In_AT."31004"[3] : Auto Mode Capability
   // // Input_Registers_In_AT."31004"[4] : Dry Mode Capability
   // // Input_Registers_In_AT."31004"[8] : Fan Direction Level Capability
   // // Input_Registers_In_AT."31004"[9] : Fan Direction Level Capability
   // // Input_Registers_In_AT."31004"[10] : Fan Direction Level Capability
   // // Input_Registers_In_AT."31004"[11] : Fan Direction Capability
   // // Input_Registers_In_AT."31004"[12] : Fan Volume Level Capability
   // // Input_Registers_In_AT."31004"[13] : Fan Volume Level Capability
   // // Input_Registers_In_AT."31004"[14] : Fan Volume Level Capability
   // // Input_Registers_In_AT."31004"[15] : Fan Volume Capability
   // // Input_Registers_In_AT."31007"[0] : Fan Mode Capability
   // // Input_Registers_In_AT."31007"[1] : Cooling Mode Capability
   // // Input_Registers_In_AT."31007"[2] : Heating Mode Capability
   // // Input_Registers_In_AT."31007"[3] : Auto Mode Capability
   // // Input_Registers_In_AT."31007"[4] : Dry Mode Capability
   // // Input_Registers_In_AT."31007"[8] : Fan Direction Level Capability
   // // Input_Registers_In_AT."31007"[9] : Fan Direction Level Capability
   // // Input_Registers_In_AT."31007"[10] : Fan Direction Level Capability
   // // Input_Registers_In_AT."31007"[11] : Fan Direction Capability
   // // Input_Registers_In_AT."31007"[12] : Fan Volume Level Capability
   // // Input_Registers_In_AT."31007"[13] : Fan Volume Level Capability
   // // Input_Registers_In_AT."31007"[14] : Fan Volume Level Capability
   // // Input_Registers_In_AT."31007"[15] : Fan Volume Capability
   // // Input_Registers_In_AT."31010"[0] : Fan Mode Capability
   // // Input_Registers_In_AT."31010"[1] : Cooling Mode Capability
   // // Input_Registers_In_AT."31010"[2] : Heating Mode Capability
   // // Input_Registers_In_AT."31010"[3] : Auto Mode Capability
   // // Input_Registers_In_AT."31010"[4] : Dry Mode Capability
   // // Input_Registers_In_AT."31010"[8] : Fan Direction Level Capability
   // // Input_Registers_In_AT."31010"[9] : Fan Direction Level Capability
   // // Input_Registers_In_AT."31010"[10] : Fan Direction Level Capability
   // // Input_Registers_In_AT."31010"[11] : Fan Direction Capability
   // // Input_Registers_In_AT."31010"[12] : Fan Volume Level Capability
   // // Input_Registers_In_AT."31010"[13] : Fan Volume Level Capability
   // // Input_Registers_In_AT."31010"[14] : Fan Volume Level Capability
   // // Input_Registers_In_AT."31010"[15] : Fan Volume Capability
   // // Input_Registers_In_AT."31013"[0] : Fan Mode Capability
   // // Input_Registers_In_AT."31013"[1] : Cooling Mode Capability
   // // Input_Registers_In_AT."31013"[2] : Heating Mode Capability
   // // Input_Registers_In_AT."31013"[3] : Auto Mode Capability
   // // Input_Registers_In_AT."31013"[4] : Dry Mode Capability
   // // Input_Registers_In_AT."31013"[8] : Fan Direction Level Capability
   // // Input_Registers_In_AT."31013"[9] : Fan Direction Level Capability
   // // Input_Registers_In_AT."31013"[10] : Fan Direction Level Capability
   // // Input_Registers_In_AT."31013"[11] : Fan Direction Capability
   // // Input_Registers_In_AT."31013"[12] : Fan Volume Level Capability
   // // Input_Registers_In_AT."31013"[13] : Fan Volume Level Capability
   // // Input_Registers_In_AT."31013"[14] : Fan Volume Level Capability
   // // Input_Registers_In_AT."31013"[15] : Fan Volume Capability
   // // Input_Registers_In_AT."31016"[0] : Fan Mode Capability
   // // Input_Registers_In_AT."31016"[1] : Cooling Mode Capability
   // // Input_Registers_In_AT."31016"[2] : Heating Mode Capability
   // // Input_Registers_In_AT."31016"[3] : Auto Mode Capability
   // // Input_Registers_In_AT."31016"[4] : Dry Mode Capability
   // // Input_Registers_In_AT."31016"[8] : Fan Direction Level Capability
   // // Input_Registers_In_AT."31016"[9] : Fan Direction Level Capability
   // // Input_Registers_In_AT."31016"[10] : Fan Direction Level Capability
   // // Input_Registers_In_AT."31016"[11] : Fan Direction Capability
   // // Input_Registers_In_AT."31016"[12] : Fan Volume Level Capability
   // // Input_Registers_In_AT."31016"[13] : Fan Volume Level Capability
   // // Input_Registers_In_AT."31016"[14] : Fan Volume Level Capability
   // // Input_Registers_In_AT."31016"[15] : Fan Volume Capability
   // // Input_Registers_In_AT."31019"[0] : Fan Mode Capability
   // // Input_Registers_In_AT."31019"[1] : Cooling Mode Capability
   // // Input_Registers_In_AT."31019"[2] : Heating Mode Capability
   // // Input_Registers_In_AT."31019"[3] : Auto Mode Capability
   // // Input_Registers_In_AT."31019"[4] : Dry Mode Capability
   // // Input_Registers_In_AT."31019"[8] : Fan Direction Level Capability
   // // Input_Registers_In_AT."31019"[9] : Fan Direction Level Capability
   // // Input_Registers_In_AT."31019"[10] : Fan Direction Level Capability
   // // Input_Registers_In_AT."31019"[11] : Fan Direction Capability
   // // Input_Registers_In_AT."31019"[12] : Fan Volume Level Capability
   // // Input_Registers_In_AT."31019"[13] : Fan Volume Level Capability
   // // Input_Registers_In_AT."31019"[14] : Fan Volume Level Capability
   // // Input_Registers_In_AT."31019"[15] : Fan Volume Capability
   // // Input_Registers_In_AT."31022"[0] : Fan Mode Capability
   // // Input_Registers_In_AT."31022"[1] : Cooling Mode Capability
   // // Input_Registers_In_AT."31022"[2] : Heating Mode Capability
   // // Input_Registers_In_AT."31022"[3] : Auto Mode Capability
   // // Input_Registers_In_AT."31022"[4] : Dry Mode Capability
   // // Input_Registers_In_AT."31022"[8] : Fan Direction Level Capability
   // // Input_Registers_In_AT."31022"[9] : Fan Direction Level Capability
   // // Input_Registers_In_AT."31022"[10] : Fan Direction Level Capability
   // // Input_Registers_In_AT."31022"[11] : Fan Direction Capability
   // // Input_Registers_In_AT."31022"[12] : Fan Volume Level Capability
   // // Input_Registers_In_AT."31022"[13] : Fan Volume Level Capability
   // // Input_Registers_In_AT."31022"[14] : Fan Volume Level Capability
   // // Input_Registers_In_AT."31022"[15] : Fan Volume Capability
   // // Input_Registers_In_AT."31025"[0] : Fan Mode Capability
   // // Input_Registers_In_AT."31025"[1] : Cooling Mode Capability
   // // Input_Registers_In_AT."31025"[2] : Heating Mode Capability
   // // Input_Registers_In_AT."31025"[3] : Auto Mode Capability
   // // Input_Registers_In_AT."31025"[4] : Dry Mode Capability
   // // Input_Registers_In_AT."31025"[8] : Fan Direction Level Capability
   // // Input_Registers_In_AT."31025"[9] : Fan Direction Level Capability
   // // Input_Registers_In_AT."31025"[10] : Fan Direction Level Capability
   // // Input_Registers_In_AT."31025"[11] : Fan Direction Capability
   // // Input_Registers_In_AT."31025"[12] : Fan Volume Level Capability
   // // Input_Registers_In_AT."31025"[13] : Fan Volume Level Capability
   // // Input_Registers_In_AT."31025"[14] : Fan Volume Level Capability
   // // Input_Registers_In_AT."31025"[15] : Fan Volume Capability
   // // Input_Registers_In_AT."31028"[0] : Fan Mode Capability
   // // Input_Registers_In_AT."31028"[1] : Cooling Mode Capability
   // // Input_Registers_In_AT."31028"[2] : Heating Mode Capability
   // // Input_Registers_In_AT."31028"[3] : Auto Mode Capability
   // // Input_Registers_In_AT."31028"[4] : Dry Mode Capability
   // // Input_Registers_In_AT."31028"[8] : Fan Direction Level Capability
   // // Input_Registers_In_AT."31028"[9] : Fan Direction Level Capability
   // // Input_Registers_In_AT."31028"[10] : Fan Direction Level Capability
   // // Input_Registers_In_AT."31028"[11] : Fan Direction Capability
   // // Input_Registers_In_AT."31028"[12] : Fan Volume Level Capability
   // // Input_Registers_In_AT."31028"[13] : Fan Volume Level Capability
   // // Input_Registers_In_AT."31028"[14] : Fan Volume Level Capability
   // // Input_Registers_In_AT."31028"[15] : Fan Volume Capability
   // // Input_Registers_In_AT."31031"[0] : Fan Mode Capability
   // // Input_Registers_In_AT."31031"[1] : Cooling Mode Capability
   // // Input_Registers_In_AT."31031"[2] : Heating Mode Capability
   // // Input_Registers_In_AT."31031"[3] : Auto Mode Capability
   // // Input_Registers_In_AT."31031"[4] : Dry Mode Capability
   // // Input_Registers_In_AT."31031"[8] : Fan Direction Level Capability
   // // Input_Registers_In_AT."31031"[9] : Fan Direction Level Capability
   // // Input_Registers_In_AT."31031"[10] : Fan Direction Level Capability
   // // Input_Registers_In_AT."31031"[11] : Fan Direction Capability
   // // Input_Registers_In_AT."31031"[12] : Fan Volume Level Capability
   // // Input_Registers_In_AT."31031"[13] : Fan Volume Level Capability
   // // Input_Registers_In_AT."31031"[14] : Fan Volume Level Capability
   // // Input_Registers_In_AT."31031"[15] : Fan Volume Capability
   // // Input_Registers_In_AT."31034"[0] : Fan Mode Capability
   // // Input_Registers_In_AT."31034"[1] : Cooling Mode Capability
   // // Input_Registers_In_AT."31034"[2] : Heating Mode Capability
   // // Input_Registers_In_AT."31034"[3] : Auto Mode Capability
   // // Input_Registers_In_AT."31034"[4] : Dry Mode Capability
   // // Input_Registers_In_AT."31034"[8] : Fan Direction Level Capability
   // // Input_Registers_In_AT."31034"[9] : Fan Direction Level Capability
   // // Input_Registers_In_AT."31034"[10] : Fan Direction Level Capability
   // // Input_Registers_In_AT."31034"[11] : Fan Direction Capability
   // // Input_Registers_In_AT."31034"[12] : Fan Volume Level Capability
   // // Input_Registers_In_AT."31034"[13] : Fan Volume Level Capability
   // // Input_Registers_In_AT."31034"[14] : Fan Volume Level Capability
   // // Input_Registers_In_AT."31034"[15] : Fan Volume Capability
   // // Input_Registers_In_AT."31037"[0] : Fan Mode Capability
   // // Input_Registers_In_AT."31037"[1] : Cooling Mode Capability
   // // Input_Registers_In_AT."31037"[2] : Heating Mode Capability
   // // Input_Registers_In_AT."31037"[3] : Auto Mode Capability
   // // Input_Registers_In_AT."31037"[4] : Dry Mode Capability
   // // Input_Registers_In_AT."31037"[8] : Fan Direction Level Capability
   // // Input_Registers_In_AT."31037"[9] : Fan Direction Level Capability
   // // Input_Registers_In_AT."31037"[10] : Fan Direction Level Capability
   // // Input_Registers_In_AT."31037"[11] : Fan Direction Capability
   // // Input_Registers_In_AT."31037"[12] : Fan Volume Level Capability
   // // Input_Registers_In_AT."31037"[13] : Fan Volume Level Capability
   // // Input_Registers_In_AT."31037"[14] : Fan Volume Level Capability
   // // Input_Registers_In_AT."31037"[15] : Fan Volume Capability
   // // Input_Registers_In_AT."31040"[0] : Fan Mode Capability
   // // Input_Registers_In_AT."31040"[1] : Cooling Mode Capability
   // // Input_Registers_In_AT."31040"[2] : Heating Mode Capability
   // // Input_Registers_In_AT."31040"[3] : Auto Mode Capability
   // // Input_Registers_In_AT."31040"[4] : Dry Mode Capability
   // // Input_Registers_In_AT."31040"[8] : Fan Direction Level Capability
   // // Input_Registers_In_AT."31040"[9] : Fan Direction Level Capability
   // // Input_Registers_In_AT."31040"[10] : Fan Direction Level Capability
   // // Input_Registers_In_AT."31040"[11] : Fan Direction Capability
   // // Input_Registers_In_AT."31040"[12] : Fan Volume Level Capability
   // // Input_Registers_In_AT."31040"[13] : Fan Volume Level Capability
   // // Input_Registers_In_AT."31040"[14] : Fan Volume Level Capability
   // // Input_Registers_In_AT."31040"[15] : Fan Volume Capability
   // // Input_Registers_In_AT."31043"[0] : Fan Mode Capability
   // // Input_Registers_In_AT."31043"[1] : Cooling Mode Capability
   // // Input_Registers_In_AT."31043"[2] : Heating Mode Capability
   // // Input_Registers_In_AT."31043"[3] : Auto Mode Capability
   // // Input_Registers_In_AT."31043"[4] : Dry Mode Capability
   // // Input_Registers_In_AT."31043"[8] : Fan Direction Level Capability
   // // Input_Registers_In_AT."31043"[9] : Fan Direction Level Capability
   // // Input_Registers_In_AT."31043"[10] : Fan Direction Level Capability
   // // Input_Registers_In_AT."31043"[11] : Fan Direction Capability
   // // Input_Registers_In_AT."31043"[12] : Fan Volume Level Capability
   // // Input_Registers_In_AT."31043"[13] : Fan Volume Level Capability
   // // Input_Registers_In_AT."31043"[14] : Fan Volume Level Capability
   // // Input_Registers_In_AT."31043"[15] : Fan Volume Capability
   // // Input_Registers_In_AT."31046"[0] : Fan Mode Capability
   // // Input_Registers_In_AT."31046"[1] : Cooling Mode Capability
   // // Input_Registers_In_AT."31046"[2] : Heating Mode Capability
   // // Input_Registers_In_AT."31046"[3] : Auto Mode Capability
   // // Input_Registers_In_AT."31046"[4] : Dry Mode Capability
   // // Input_Registers_In_AT."31046"[8] : Fan Direction Level Capability
   // // Input_Registers_In_AT."31046"[9] : Fan Direction Level Capability
   // // Input_Registers_In_AT."31046"[10] : Fan Direction Level Capability
   // // Input_Registers_In_AT."31046"[11] : Fan Direction Capability
   // // Input_Registers_In_AT."31046"[12] : Fan Volume Level Capability
   // // Input_Registers_In_AT."31046"[13] : Fan Volume Level Capability
   // // Input_Registers_In_AT."31046"[14] : Fan Volume Level Capability
   // // Input_Registers_In_AT."31046"[15] : Fan Volume Capability
   // // Input_Registers_In_AT."32001"[0] : OnOff Status
   // // Input_Registers_In_AT."32001"[2] : Forced off status
   // // Input_Registers_In_AT."32001"[8] : Fan direction
   // // Input_Registers_In_AT."32001"[9] : Fan direction
   // // Input_Registers_In_AT."32001"[10] : Fan direction
   // // Input_Registers_In_AT."32001"[12] : Fan volume
   // // Input_Registers_In_AT."32001"[13] : Fan volume
   // // Input_Registers_In_AT."32001"[14] : Fan volume
   // // Input_Registers_In_AT."32002"[0] : Operation mode
   // // Input_Registers_In_AT."32002"[1] : Operation mode
   // // Input_Registers_In_AT."32002"[2] : Operation mode
   // // Input_Registers_In_AT."32002"[3] : Operation mode
   // // Input_Registers_In_AT."32002"[4] : Filter sign status
   // // Input_Registers_In_AT."32002"[5] : Filter sign status
   // // Input_Registers_In_AT."32002"[6] : Filter sign status
   // // Input_Registers_In_AT."32002"[7] : Filter sign status
   // // Input_Registers_In_AT."32002"[8] : Operation status
   // // Input_Registers_In_AT."32002"[9] : Operation status
   // // Input_Registers_In_AT."32002"[10] : Operation status
   // // Input_Registers_In_AT."32002"[11] : Operation status
   // // Input_Registers_In_AT."32002"[14] : Cool/Heat Master
   // // Input_Registers_In_AT."32002"[15] : Cool/Heat Master
   // // Input_Registers_In_AT."32003"[15] : Signed Bit
   // // Input_Registers_In_AT."32004"[0] : Error code mapping value1
   // // Input_Registers_In_AT."32004"[1] : Error code mapping value1
   // // Input_Registers_In_AT."32004"[2] : Error code mapping value1
   // // Input_Registers_In_AT."32004"[3] : Error code mapping value1
   // // Input_Registers_In_AT."32004"[4] : Error code mapping value2
   // // Input_Registers_In_AT."32004"[5] : Error code mapping value2
   // // Input_Registers_In_AT."32004"[6] : Error code mapping value2
   // // Input_Registers_In_AT."32004"[7] : Error code mapping value2
   // // Input_Registers_In_AT."32004"[8] : Malfunction
   // // Input_Registers_In_AT."32004"[9] : Warning
   // // Input_Registers_In_AT."32004"[10] : Operation status
   // // Input_Registers_In_AT."32005"[15] : Signed Bit
   // // Input_Registers_In_AT."32006"[8] : Indoor unit temperature sensor error
   // // Input_Registers_In_AT."32006"[15] : Indoor unit temperature sensor data received
   // // Input_Registers_In_AT."32007"[0] : OnOff Status
   // // Input_Registers_In_AT."32007"[2] : Forced off status
   // // Input_Registers_In_AT."32007"[8] : Fan direction
   // // Input_Registers_In_AT."32007"[9] : Fan direction
   // // Input_Registers_In_AT."32007"[10] : Fan direction
   // // Input_Registers_In_AT."32007"[12] : Fan volume
   // // Input_Registers_In_AT."32007"[13] : Fan volume
   // // Input_Registers_In_AT."32007"[14] : Fan volume
   // // Input_Registers_In_AT."32008"[0] : Operation mode
   // // Input_Registers_In_AT."32008"[1] : Operation mode
   // // Input_Registers_In_AT."32008"[2] : Operation mode
   // // Input_Registers_In_AT."32008"[3] : Operation mode
   // // Input_Registers_In_AT."32008"[4] : Filter sign status
   // // Input_Registers_In_AT."32008"[5] : Filter sign status
   // // Input_Registers_In_AT."32008"[6] : Filter sign status
   // // Input_Registers_In_AT."32008"[7] : Filter sign status
   // // Input_Registers_In_AT."32008"[8] : Operation status
   // // Input_Registers_In_AT."32008"[9] : Operation status
   // // Input_Registers_In_AT."32008"[10] : Operation status
   // // Input_Registers_In_AT."32008"[11] : Operation status
   // // Input_Registers_In_AT."32008"[14] : Cool/Heat Master
   // // Input_Registers_In_AT."32008"[15] : Cool/Heat Master
   // // Input_Registers_In_AT."32009"[15] : Signed Bit
   // // Input_Registers_In_AT."32010"[0] : Error code mapping value1
   // // Input_Registers_In_AT."32010"[1] : Error code mapping value1
   // // Input_Registers_In_AT."32010"[2] : Error code mapping value1
   // // Input_Registers_In_AT."32010"[3] : Error code mapping value1
   // // Input_Registers_In_AT."32010"[4] : Error code mapping value2
   // // Input_Registers_In_AT."32010"[5] : Error code mapping value2
   // // Input_Registers_In_AT."32010"[6] : Error code mapping value2
   // // Input_Registers_In_AT."32010"[7] : Error code mapping value2
   // // Input_Registers_In_AT."32010"[8] : Malfunction
   // // Input_Registers_In_AT."32010"[9] : Warning
   // // Input_Registers_In_AT."32010"[10] : Operation status
   // // Input_Registers_In_AT."32011"[15] : Signed Bit
   // // Input_Registers_In_AT."32012"[8] : Indoor unit temperature sensor error
   // // Input_Registers_In_AT."32012"[15] : Indoor unit temperature sensor data received
   // // Input_Registers_In_AT."32013"[0] : OnOff Status
   // // Input_Registers_In_AT."32013"[2] : Forced off status
   // // Input_Registers_In_AT."32013"[8] : Fan direction
   // // Input_Registers_In_AT."32013"[9] : Fan direction
   // // Input_Registers_In_AT."32013"[10] : Fan direction
   // // Input_Registers_In_AT."32013"[12] : Fan volume
   // // Input_Registers_In_AT."32013"[13] : Fan volume
   // // Input_Registers_In_AT."32013"[14] : Fan volume
   // // Input_Registers_In_AT."32014"[0] : Operation mode
   // // Input_Registers_In_AT."32014"[1] : Operation mode
   // // Input_Registers_In_AT."32014"[2] : Operation mode
   // // Input_Registers_In_AT."32014"[3] : Operation mode
   // // Input_Registers_In_AT."32014"[4] : Filter sign status
   // // Input_Registers_In_AT."32014"[5] : Filter sign status
   // // Input_Registers_In_AT."32014"[6] : Filter sign status
   // // Input_Registers_In_AT."32014"[7] : Filter sign status
   // // Input_Registers_In_AT."32014"[8] : Operation status
   // // Input_Registers_In_AT."32014"[9] : Operation status
   // // Input_Registers_In_AT."32014"[10] : Operation status
   // // Input_Registers_In_AT."32014"[11] : Operation status
   // // Input_Registers_In_AT."32014"[14] : Cool/Heat Master
   // // Input_Registers_In_AT."32014"[15] : Cool/Heat Master
   // // Input_Registers_In_AT."32015"[15] : Signed Bit
   // // Input_Registers_In_AT."32016"[0] : Error code mapping value1
   // // Input_Registers_In_AT."32016"[1] : Error code mapping value1
   // // Input_Registers_In_AT."32016"[2] : Error code mapping value1
   // // Input_Registers_In_AT."32016"[3] : Error code mapping value1
   // // Input_Registers_In_AT."32016"[4] : Error code mapping value2
   // // Input_Registers_In_AT."32016"[5] : Error code mapping value2
   // // Input_Registers_In_AT."32016"[6] : Error code mapping value2
   // // Input_Registers_In_AT."32016"[7] : Error code mapping value2
   // // Input_Registers_In_AT."32016"[8] : Malfunction
   // // Input_Registers_In_AT."32016"[9] : Warning
   // // Input_Registers_In_AT."32016"[10] : Operation status
   // // Input_Registers_In_AT."32017"[15] : Signed Bit
   // // Input_Registers_In_AT."32018"[8] : Indoor unit temperature sensor error
   // // Input_Registers_In_AT."32018"[15] : Indoor unit temperature sensor data received
   // // Input_Registers_In_AT."32019"[0] : OnOff Status
   // // Input_Registers_In_AT."32019"[2] : Forced off status
   // // Input_Registers_In_AT."32019"[8] : Fan direction
   // // Input_Registers_In_AT."32019"[9] : Fan direction
   // // Input_Registers_In_AT."32019"[10] : Fan direction
   // // Input_Registers_In_AT."32019"[12] : Fan volume
   // // Input_Registers_In_AT."32019"[13] : Fan volume
   // // Input_Registers_In_AT."32019"[14] : Fan volume
   // // Input_Registers_In_AT."32020"[0] : Operation mode
   // // Input_Registers_In_AT."32020"[1] : Operation mode
   // // Input_Registers_In_AT."32020"[2] : Operation mode
   // // Input_Registers_In_AT."32020"[3] : Operation mode
   // // Input_Registers_In_AT."32020"[4] : Filter sign status
   // // Input_Registers_In_AT."32020"[5] : Filter sign status
   // // Input_Registers_In_AT."32020"[6] : Filter sign status
   // // Input_Registers_In_AT."32020"[7] : Filter sign status
   // // Input_Registers_In_AT."32020"[8] : Operation status
   // // Input_Registers_In_AT."32020"[9] : Operation status
   // // Input_Registers_In_AT."32020"[10] : Operation status
   // // Input_Registers_In_AT."32020"[11] : Operation status
   // // Input_Registers_In_AT."32020"[14] : Cool/Heat Master
   // // Input_Registers_In_AT."32020"[15] : Cool/Heat Master
   // // Input_Registers_In_AT."32021"[15] : Signed Bit
   // // Input_Registers_In_AT."32022"[0] : Error code mapping value1
   // // Input_Registers_In_AT."32022"[1] : Error code mapping value1
   // // Input_Registers_In_AT."32022"[2] : Error code mapping value1
   // // Input_Registers_In_AT."32022"[3] : Error code mapping value1
   // // Input_Registers_In_AT."32022"[4] : Error code mapping value2
   // // Input_Registers_In_AT."32022"[5] : Error code mapping value2
   // // Input_Registers_In_AT."32022"[6] : Error code mapping value2
   // // Input_Registers_In_AT."32022"[7] : Error code mapping value2
   // // Input_Registers_In_AT."32022"[8] : Malfunction
   // // Input_Registers_In_AT."32022"[9] : Warning
   // // Input_Registers_In_AT."32022"[10] : Operation status
   // // Input_Registers_In_AT."32023"[15] : Signed Bit
   // // Input_Registers_In_AT."32024"[8] : Indoor unit temperature sensor error
   // // Input_Registers_In_AT."32024"[15] : Indoor unit temperature sensor data received
   // // Input_Registers_In_AT."32025"[0] : OnOff Status
   // // Input_Registers_In_AT."32025"[2] : Forced off status
   // // Input_Registers_In_AT."32025"[8] : Fan direction
   // // Input_Registers_In_AT."32025"[9] : Fan direction
   // // Input_Registers_In_AT."32025"[10] : Fan direction
   // // Input_Registers_In_AT."32025"[12] : Fan volume
   // // Input_Registers_In_AT."32025"[13] : Fan volume
   // // Input_Registers_In_AT."32025"[14] : Fan volume
   // // Input_Registers_In_AT."32026"[0] : Operation mode
   // // Input_Registers_In_AT."32026"[1] : Operation mode
   // // Input_Registers_In_AT."32026"[2] : Operation mode
   // // Input_Registers_In_AT."32026"[3] : Operation mode
   // // Input_Registers_In_AT."32026"[4] : Filter sign status
   // // Input_Registers_In_AT."32026"[5] : Filter sign status
   // // Input_Registers_In_AT."32026"[6] : Filter sign status
   // // Input_Registers_In_AT."32026"[7] : Filter sign status
   // // Input_Registers_In_AT."32026"[8] : Operation status
   // // Input_Registers_In_AT."32026"[9] : Operation status
   // // Input_Registers_In_AT."32026"[10] : Operation status
   // // Input_Registers_In_AT."32026"[11] : Operation status
   // // Input_Registers_In_AT."32026"[14] : Cool/Heat Master
   // // Input_Registers_In_AT."32026"[15] : Cool/Heat Master
   // // Input_Registers_In_AT."32027"[15] : Signed Bit
   // // Input_Registers_In_AT."32028"[0] : Error code mapping value1
   // // Input_Registers_In_AT."32028"[1] : Error code mapping value1
   // // Input_Registers_In_AT."32028"[2] : Error code mapping value1
   // // Input_Registers_In_AT."32028"[3] : Error code mapping value1
   // // Input_Registers_In_AT."32028"[4] : Error code mapping value2
   // // Input_Registers_In_AT."32028"[5] : Error code mapping value2
   // // Input_Registers_In_AT."32028"[6] : Error code mapping value2
   // // Input_Registers_In_AT."32028"[7] : Error code mapping value2
   // // Input_Registers_In_AT."32028"[8] : Malfunction
   // // Input_Registers_In_AT."32028"[9] : Warning
   // // Input_Registers_In_AT."32028"[10] : Operation status
   // // Input_Registers_In_AT."32029"[15] : Signed Bit
   // // Input_Registers_In_AT."32030"[8] : Indoor unit temperature sensor error
   // // Input_Registers_In_AT."32030"[15] : Indoor unit temperature sensor data received
   // // Input_Registers_In_AT."32031"[0] : OnOff Status
   // // Input_Registers_In_AT."32031"[2] : Forced off status
   // // Input_Registers_In_AT."32031"[8] : Fan direction
   // // Input_Registers_In_AT."32031"[9] : Fan direction
   // // Input_Registers_In_AT."32031"[10] : Fan direction
   // // Input_Registers_In_AT."32031"[12] : Fan volume
   // // Input_Registers_In_AT."32031"[13] : Fan volume
   // // Input_Registers_In_AT."32031"[14] : Fan volume
   // // Input_Registers_In_AT."32032"[0] : Operation mode
   // // Input_Registers_In_AT."32032"[1] : Operation mode
   // // Input_Registers_In_AT."32032"[2] : Operation mode
   // // Input_Registers_In_AT."32032"[3] : Operation mode
   // // Input_Registers_In_AT."32032"[4] : Filter sign status
   // // Input_Registers_In_AT."32032"[5] : Filter sign status
   // // Input_Registers_In_AT."32032"[6] : Filter sign status
   // // Input_Registers_In_AT."32032"[7] : Filter sign status
   // // Input_Registers_In_AT."32032"[8] : Operation status
   // // Input_Registers_In_AT."32032"[9] : Operation status
   // // Input_Registers_In_AT."32032"[10] : Operation status
   // // Input_Registers_In_AT."32032"[11] : Operation status
   // // Input_Registers_In_AT."32032"[14] : Cool/Heat Master
   // // Input_Registers_In_AT."32032"[15] : Cool/Heat Master
   // // Input_Registers_In_AT."32033"[15] : Signed Bit
   // // Input_Registers_In_AT."32034"[0] : Error code mapping value1
   // // Input_Registers_In_AT."32034"[1] : Error code mapping value1
   // // Input_Registers_In_AT."32034"[2] : Error code mapping value1
   // // Input_Registers_In_AT."32034"[3] : Error code mapping value1
   // // Input_Registers_In_AT."32034"[4] : Error code mapping value2
   // // Input_Registers_In_AT."32034"[5] : Error code mapping value2
   // // Input_Registers_In_AT."32034"[6] : Error code mapping value2
   // // Input_Registers_In_AT."32034"[7] : Error code mapping value2
   // // Input_Registers_In_AT."32034"[8] : Malfunction
   // // Input_Registers_In_AT."32034"[9] : Warning
   // // Input_Registers_In_AT."32034"[10] : Operation status
   // // Input_Registers_In_AT."32035"[15] : Signed Bit
   // // Input_Registers_In_AT."32036"[8] : Indoor unit temperature sensor error
   // // Input_Registers_In_AT."32036"[15] : Indoor unit temperature sensor data received
   // // Input_Registers_In_AT."32037"[0] : OnOff Status
   // // Input_Registers_In_AT."32037"[2] : Forced off status
   // // Input_Registers_In_AT."32037"[8] : Fan direction
   // // Input_Registers_In_AT."32037"[9] : Fan direction
   // // Input_Registers_In_AT."32037"[10] : Fan direction
   // // Input_Registers_In_AT."32037"[12] : Fan volume
   // // Input_Registers_In_AT."32037"[13] : Fan volume
   // // Input_Registers_In_AT."32037"[14] : Fan volume
   // // Input_Registers_In_AT."32038"[0] : Operation mode
   // // Input_Registers_In_AT."32038"[1] : Operation mode
   // // Input_Registers_In_AT."32038"[2] : Operation mode
   // // Input_Registers_In_AT."32038"[3] : Operation mode
   // // Input_Registers_In_AT."32038"[4] : Filter sign status
   // // Input_Registers_In_AT."32038"[5] : Filter sign status
   // // Input_Registers_In_AT."32038"[6] : Filter sign status
   // // Input_Registers_In_AT."32038"[7] : Filter sign status
   // // Input_Registers_In_AT."32038"[8] : Operation status
   // // Input_Registers_In_AT."32038"[9] : Operation status
   // // Input_Registers_In_AT."32038"[10] : Operation status
   // // Input_Registers_In_AT."32038"[11] : Operation status
   // // Input_Registers_In_AT."32038"[14] : Cool/Heat Master
   // // Input_Registers_In_AT."32038"[15] : Cool/Heat Master
   // // Input_Registers_In_AT."32039"[15] : Signed Bit
   // // Input_Registers_In_AT."32040"[0] : Error code mapping value1
   // // Input_Registers_In_AT."32040"[1] : Error code mapping value1
   // // Input_Registers_In_AT."32040"[2] : Error code mapping value1
   // // Input_Registers_In_AT."32040"[3] : Error code mapping value1
   // // Input_Registers_In_AT."32040"[4] : Error code mapping value2
   // // Input_Registers_In_AT."32040"[5] : Error code mapping value2
   // // Input_Registers_In_AT."32040"[6] : Error code mapping value2
   // // Input_Registers_In_AT."32040"[7] : Error code mapping value2
   // // Input_Registers_In_AT."32040"[8] : Malfunction
   // // Input_Registers_In_AT."32040"[9] : Warning
   // // Input_Registers_In_AT."32040"[10] : Operation status
   // // Input_Registers_In_AT."32041"[15] : Signed Bit
   // // Input_Registers_In_AT."32042"[8] : Indoor unit temperature sensor error
   // // Input_Registers_In_AT."32042"[15] : Indoor unit temperature sensor data received
   // // Input_Registers_In_AT."32043"[0] : OnOff Status
   // // Input_Registers_In_AT."32043"[2] : Forced off status
   // // Input_Registers_In_AT."32043"[8] : Fan direction
   // // Input_Registers_In_AT."32043"[9] : Fan direction
   // // Input_Registers_In_AT."32043"[10] : Fan direction
   // // Input_Registers_In_AT."32043"[12] : Fan volume
   // // Input_Registers_In_AT."32043"[13] : Fan volume
   // // Input_Registers_In_AT."32043"[14] : Fan volume
   // // Input_Registers_In_AT."32044"[0] : Operation mode
   // // Input_Registers_In_AT."32044"[1] : Operation mode
   // // Input_Registers_In_AT."32044"[2] : Operation mode
   // // Input_Registers_In_AT."32044"[3] : Operation mode
   // // Input_Registers_In_AT."32044"[4] : Filter sign status
   // // Input_Registers_In_AT."32044"[5] : Filter sign status
   // // Input_Registers_In_AT."32044"[6] : Filter sign status
   // // Input_Registers_In_AT."32044"[7] : Filter sign status
   // // Input_Registers_In_AT."32044"[8] : Operation status
   // // Input_Registers_In_AT."32044"[9] : Operation status
   // // Input_Registers_In_AT."32044"[10] : Operation status
   // // Input_Registers_In_AT."32044"[11] : Operation status
   // // Input_Registers_In_AT."32044"[14] : Cool/Heat Master
   // // Input_Registers_In_AT."32044"[15] : Cool/Heat Master
   // // Input_Registers_In_AT."32045"[15] : Signed Bit
   // // Input_Registers_In_AT."32046"[0] : Error code mapping value1
   // // Input_Registers_In_AT."32046"[1] : Error code mapping value1
   // // Input_Registers_In_AT."32046"[2] : Error code mapping value1
   // // Input_Registers_In_AT."32046"[3] : Error code mapping value1
   // // Input_Registers_In_AT."32046"[4] : Error code mapping value2
   // // Input_Registers_In_AT."32046"[5] : Error code mapping value2
   // // Input_Registers_In_AT."32046"[6] : Error code mapping value2
   // // Input_Registers_In_AT."32046"[7] : Error code mapping value2
   // // Input_Registers_In_AT."32046"[8] : Malfunction
   // // Input_Registers_In_AT."32046"[9] : Warning
   // // Input_Registers_In_AT."32046"[10] : Operation status
   // // Input_Registers_In_AT."32047"[15] : Signed Bit
   // // Input_Registers_In_AT."32048"[8] : Indoor unit temperature sensor error
   // // Input_Registers_In_AT."32048"[15] : Indoor unit temperature sensor data received
   // // Input_Registers_In_AT."32049"[0] : OnOff Status
   // // Input_Registers_In_AT."32049"[2] : Forced off status
   // // Input_Registers_In_AT."32049"[8] : Fan direction
   // // Input_Registers_In_AT."32049"[9] : Fan direction
   // // Input_Registers_In_AT."32049"[10] : Fan direction
   // // Input_Registers_In_AT."32049"[12] : Fan volume
   // // Input_Registers_In_AT."32049"[13] : Fan volume
   // // Input_Registers_In_AT."32049"[14] : Fan volume
   // // Input_Registers_In_AT."32050"[0] : Operation mode
   // // Input_Registers_In_AT."32050"[1] : Operation mode
   // // Input_Registers_In_AT."32050"[2] : Operation mode
   // // Input_Registers_In_AT."32050"[3] : Operation mode
   // // Input_Registers_In_AT."32050"[4] : Filter sign status
   // // Input_Registers_In_AT."32050"[5] : Filter sign status
   // // Input_Registers_In_AT."32050"[6] : Filter sign status
   // // Input_Registers_In_AT."32050"[7] : Filter sign status
   // // Input_Registers_In_AT."32050"[8] : Operation status
   // // Input_Registers_In_AT."32050"[9] : Operation status
   // // Input_Registers_In_AT."32050"[10] : Operation status
   // // Input_Registers_In_AT."32050"[11] : Operation status
   // // Input_Registers_In_AT."32050"[14] : Cool/Heat Master
   // // Input_Registers_In_AT."32050"[15] : Cool/Heat Master
   // // Input_Registers_In_AT."32051"[15] : Signed Bit
   // // Input_Registers_In_AT."32052"[0] : Error code mapping value1
   // // Input_Registers_In_AT."32052"[1] : Error code mapping value1
   // // Input_Registers_In_AT."32052"[2] : Error code mapping value1
   // // Input_Registers_In_AT."32052"[3] : Error code mapping value1
   // // Input_Registers_In_AT."32052"[4] : Error code mapping value2
   // // Input_Registers_In_AT."32052"[5] : Error code mapping value2
   // // Input_Registers_In_AT."32052"[6] : Error code mapping value2
   // // Input_Registers_In_AT."32052"[7] : Error code mapping value2
   // // Input_Registers_In_AT."32052"[8] : Malfunction
   // // Input_Registers_In_AT."32052"[9] : Warning
   // // Input_Registers_In_AT."32052"[10] : Operation status
   // // Input_Registers_In_AT."32053"[15] : Signed Bit
   // // Input_Registers_In_AT."32054"[8] : Indoor unit temperature sensor error
   // // Input_Registers_In_AT."32054"[15] : Indoor unit temperature sensor data received
   // // Input_Registers_In_AT."32055"[0] : OnOff Status
   // // Input_Registers_In_AT."32055"[2] : Forced off status
   // // Input_Registers_In_AT."32055"[8] : Fan direction
   // // Input_Registers_In_AT."32055"[9] : Fan direction
   // // Input_Registers_In_AT."32055"[10] : Fan direction
   // // Input_Registers_In_AT."32055"[12] : Fan volume
   // // Input_Registers_In_AT."32055"[13] : Fan volume
   // // Input_Registers_In_AT."32055"[14] : Fan volume
   // // Input_Registers_In_AT."32056"[0] : Operation mode
   // // Input_Registers_In_AT."32056"[1] : Operation mode
   // // Input_Registers_In_AT."32056"[2] : Operation mode
   // // Input_Registers_In_AT."32056"[3] : Operation mode
   // // Input_Registers_In_AT."32056"[4] : Filter sign status
   // // Input_Registers_In_AT."32056"[5] : Filter sign status
   // // Input_Registers_In_AT."32056"[6] : Filter sign status
   // // Input_Registers_In_AT."32056"[7] : Filter sign status
   // // Input_Registers_In_AT."32056"[8] : Operation status
   // // Input_Registers_In_AT."32056"[9] : Operation status
   // // Input_Registers_In_AT."32056"[10] : Operation status
   // // Input_Registers_In_AT."32056"[11] : Operation status
   // // Input_Registers_In_AT."32056"[14] : Cool/Heat Master
   // // Input_Registers_In_AT."32056"[15] : Cool/Heat Master
   // // Input_Registers_In_AT."32057"[15] : Signed Bit
   // // Input_Registers_In_AT."32058"[0] : Error code mapping value1
   // // Input_Registers_In_AT."32058"[1] : Error code mapping value1
   // // Input_Registers_In_AT."32058"[2] : Error code mapping value1
   // // Input_Registers_In_AT."32058"[3] : Error code mapping value1
   // // Input_Registers_In_AT."32058"[4] : Error code mapping value2
   // // Input_Registers_In_AT."32058"[5] : Error code mapping value2
   // // Input_Registers_In_AT."32058"[6] : Error code mapping value2
   // // Input_Registers_In_AT."32058"[7] : Error code mapping value2
   // // Input_Registers_In_AT."32058"[8] : Malfunction
   // // Input_Registers_In_AT."32058"[9] : Warning
   // // Input_Registers_In_AT."32058"[10] : Operation status
   // // Input_Registers_In_AT."32059"[15] : Signed Bit
   // // Input_Registers_In_AT."32060"[8] : Indoor unit temperature sensor error
   // // Input_Registers_In_AT."32060"[15] : Indoor unit temperature sensor data received
   // // Input_Registers_In_AT."32061"[0] : OnOff Status
   // // Input_Registers_In_AT."32061"[2] : Forced off status
   // // Input_Registers_In_AT."32061"[8] : Fan direction
   // // Input_Registers_In_AT."32061"[9] : Fan direction
   // // Input_Registers_In_AT."32061"[10] : Fan direction
   // // Input_Registers_In_AT."32061"[12] : Fan volume
   // // Input_Registers_In_AT."32061"[13] : Fan volume
   // // Input_Registers_In_AT."32061"[14] : Fan volume
   // // Input_Registers_In_AT."32062"[0] : Operation mode
   // // Input_Registers_In_AT."32062"[1] : Operation mode
   // // Input_Registers_In_AT."32062"[2] : Operation mode
   // // Input_Registers_In_AT."32062"[3] : Operation mode
   // // Input_Registers_In_AT."32062"[4] : Filter sign status
   // // Input_Registers_In_AT."32062"[5] : Filter sign status
   // // Input_Registers_In_AT."32062"[6] : Filter sign status
   // // Input_Registers_In_AT."32062"[7] : Filter sign status
   // // Input_Registers_In_AT."32062"[8] : Operation status
   // // Input_Registers_In_AT."32062"[9] : Operation status
   // // Input_Registers_In_AT."32062"[10] : Operation status
   // // Input_Registers_In_AT."32062"[11] : Operation status
   // // Input_Registers_In_AT."32062"[14] : Cool/Heat Master
   // // Input_Registers_In_AT."32062"[15] : Cool/Heat Master
   // // Input_Registers_In_AT."32063"[15] : Signed Bit
   // // Input_Registers_In_AT."32064"[0] : Error code mapping value1
   // // Input_Registers_In_AT."32064"[1] : Error code mapping value1
   // // Input_Registers_In_AT."32064"[2] : Error code mapping value1
   // // Input_Registers_In_AT."32064"[3] : Error code mapping value1
   // // Input_Registers_In_AT."32064"[4] : Error code mapping value2
   // // Input_Registers_In_AT."32064"[5] : Error code mapping value2
   // // Input_Registers_In_AT."32064"[6] : Error code mapping value2
   // // Input_Registers_In_AT."32064"[7] : Error code mapping value2
   // // Input_Registers_In_AT."32064"[8] : Malfunction
   // // Input_Registers_In_AT."32064"[9] : Warning
   // // Input_Registers_In_AT."32064"[10] : Operation status
   // // Input_Registers_In_AT."32065"[15] : Signed Bit
   // // Input_Registers_In_AT."32066"[8] : Indoor unit temperature sensor error
   // // Input_Registers_In_AT."32066"[15] : Indoor unit temperature sensor data received
   // // Input_Registers_In_AT."32067"[0] : OnOff Status
   // // Input_Registers_In_AT."32067"[2] : Forced off status
   // // Input_Registers_In_AT."32067"[8] : Fan direction
   // // Input_Registers_In_AT."32067"[9] : Fan direction
   // // Input_Registers_In_AT."32067"[10] : Fan direction
   // // Input_Registers_In_AT."32067"[12] : Fan volume
   // // Input_Registers_In_AT."32067"[13] : Fan volume
   // // Input_Registers_In_AT."32067"[14] : Fan volume
   // // Input_Registers_In_AT."32068"[0] : Operation mode
   // // Input_Registers_In_AT."32068"[1] : Operation mode
   // // Input_Registers_In_AT."32068"[2] : Operation mode
   // // Input_Registers_In_AT."32068"[3] : Operation mode
   // // Input_Registers_In_AT."32068"[4] : Filter sign status
   // // Input_Registers_In_AT."32068"[5] : Filter sign status
   // // Input_Registers_In_AT."32068"[6] : Filter sign status
   // // Input_Registers_In_AT."32068"[7] : Filter sign status
   // // Input_Registers_In_AT."32068"[8] : Operation status
   // // Input_Registers_In_AT."32068"[9] : Operation status
   // // Input_Registers_In_AT."32068"[10] : Operation status
   // // Input_Registers_In_AT."32068"[11] : Operation status
   // // Input_Registers_In_AT."32068"[14] : Cool/Heat Master
   // // Input_Registers_In_AT."32068"[15] : Cool/Heat Master
   // // Input_Registers_In_AT."32069"[15] : Signed Bit
   // // Input_Registers_In_AT."32070"[0] : Error code mapping value1
   // // Input_Registers_In_AT."32070"[1] : Error code mapping value1
   // // Input_Registers_In_AT."32070"[2] : Error code mapping value1
   // // Input_Registers_In_AT."32070"[3] : Error code mapping value1
   // // Input_Registers_In_AT."32070"[4] : Error code mapping value2
   // // Input_Registers_In_AT."32070"[5] : Error code mapping value2
   // // Input_Registers_In_AT."32070"[6] : Error code mapping value2
   // // Input_Registers_In_AT."32070"[7] : Error code mapping value2
   // // Input_Registers_In_AT."32070"[8] : Malfunction
   // // Input_Registers_In_AT."32070"[9] : Warning
   // // Input_Registers_In_AT."32070"[10] : Operation status
   // // Input_Registers_In_AT."32071"[15] : Signed Bit
   // // Input_Registers_In_AT."32072"[8] : Indoor unit temperature sensor error
   // // Input_Registers_In_AT."32072"[15] : Indoor unit temperature sensor data received
   // // Input_Registers_In_AT."32073"[0] : OnOff Status
   // // Input_Registers_In_AT."32073"[2] : Forced off status
   // // Input_Registers_In_AT."32073"[8] : Fan direction
   // // Input_Registers_In_AT."32073"[9] : Fan direction
   // // Input_Registers_In_AT."32073"[10] : Fan direction
   // // Input_Registers_In_AT."32073"[12] : Fan volume
   // // Input_Registers_In_AT."32073"[13] : Fan volume
   // // Input_Registers_In_AT."32073"[14] : Fan volume
   // // Input_Registers_In_AT."32074"[0] : Operation mode
   // // Input_Registers_In_AT."32074"[1] : Operation mode
   // // Input_Registers_In_AT."32074"[2] : Operation mode
   // // Input_Registers_In_AT."32074"[3] : Operation mode
   // // Input_Registers_In_AT."32074"[4] : Filter sign status
   // // Input_Registers_In_AT."32074"[5] : Filter sign status
   // // Input_Registers_In_AT."32074"[6] : Filter sign status
   // // Input_Registers_In_AT."32074"[7] : Filter sign status
   // // Input_Registers_In_AT."32074"[8] : Operation status
   // // Input_Registers_In_AT."32074"[9] : Operation status
   // // Input_Registers_In_AT."32074"[10] : Operation status
   // // Input_Registers_In_AT."32074"[11] : Operation status
   // // Input_Registers_In_AT."32074"[14] : Cool/Heat Master
   // // Input_Registers_In_AT."32074"[15] : Cool/Heat Master
   // // Input_Registers_In_AT."32075"[15] : Signed Bit
   // // Input_Registers_In_AT."32076"[0] : Error code mapping value1
   // // Input_Registers_In_AT."32076"[1] : Error code mapping value1
   // // Input_Registers_In_AT."32076"[2] : Error code mapping value1
   // // Input_Registers_In_AT."32076"[3] : Error code mapping value1
   // // Input_Registers_In_AT."32076"[4] : Error code mapping value2
   // // Input_Registers_In_AT."32076"[5] : Error code mapping value2
   // // Input_Registers_In_AT."32076"[6] : Error code mapping value2
   // // Input_Registers_In_AT."32076"[7] : Error code mapping value2
   // // Input_Registers_In_AT."32076"[8] : Malfunction
   // // Input_Registers_In_AT."32076"[9] : Warning
   // // Input_Registers_In_AT."32076"[10] : Operation status
   // // Input_Registers_In_AT."32077"[15] : Signed Bit
   // // Input_Registers_In_AT."32078"[8] : Indoor unit temperature sensor error
   // // Input_Registers_In_AT."32078"[15] : Indoor unit temperature sensor data received
   // // Input_Registers_In_AT."32079"[0] : OnOff Status
   // // Input_Registers_In_AT."32079"[2] : Forced off status
   // // Input_Registers_In_AT."32079"[8] : Fan direction
   // // Input_Registers_In_AT."32079"[9] : Fan direction
   // // Input_Registers_In_AT."32079"[10] : Fan direction
   // // Input_Registers_In_AT."32079"[12] : Fan volume
   // // Input_Registers_In_AT."32079"[13] : Fan volume
   // // Input_Registers_In_AT."32079"[14] : Fan volume
   // // Input_Registers_In_AT."32080"[0] : Operation mode
   // // Input_Registers_In_AT."32080"[1] : Operation mode
   // // Input_Registers_In_AT."32080"[2] : Operation mode
   // // Input_Registers_In_AT."32080"[3] : Operation mode
   // // Input_Registers_In_AT."32080"[4] : Filter sign status
   // // Input_Registers_In_AT."32080"[5] : Filter sign status
   // // Input_Registers_In_AT."32080"[6] : Filter sign status
   // // Input_Registers_In_AT."32080"[7] : Filter sign status
   // // Input_Registers_In_AT."32080"[8] : Operation status
   // // Input_Registers_In_AT."32080"[9] : Operation status
   // // Input_Registers_In_AT."32080"[10] : Operation status
   // // Input_Registers_In_AT."32080"[11] : Operation status
   // // Input_Registers_In_AT."32080"[14] : Cool/Heat Master
   // // Input_Registers_In_AT."32080"[15] : Cool/Heat Master
   // // Input_Registers_In_AT."32081"[15] : Signed Bit
   // // Input_Registers_In_AT."32082"[0] : Error code mapping value1
   // // Input_Registers_In_AT."32082"[1] : Error code mapping value1
   // // Input_Registers_In_AT."32082"[2] : Error code mapping value1
   // // Input_Registers_In_AT."32082"[3] : Error code mapping value1
   // // Input_Registers_In_AT."32082"[4] : Error code mapping value2
   // // Input_Registers_In_AT."32082"[5] : Error code mapping value2
   // // Input_Registers_In_AT."32082"[6] : Error code mapping value2
   // // Input_Registers_In_AT."32082"[7] : Error code mapping value2
   // // Input_Registers_In_AT."32082"[8] : Malfunction
   // // Input_Registers_In_AT."32082"[9] : Warning
   // // Input_Registers_In_AT."32082"[10] : Operation status
   // // Input_Registers_In_AT."32083"[15] : Signed Bit
   // // Input_Registers_In_AT."32084"[8] : Indoor unit temperature sensor error
   // // Input_Registers_In_AT."32084"[15] : Indoor unit temperature sensor data received
   // // Input_Registers_In_AT."32085"[0] : OnOff Status
   // // Input_Registers_In_AT."32085"[2] : Forced off status
   // // Input_Registers_In_AT."32085"[8] : Fan direction
   // // Input_Registers_In_AT."32085"[9] : Fan direction
   // // Input_Registers_In_AT."32085"[10] : Fan direction
   // // Input_Registers_In_AT."32085"[12] : Fan volume
   // // Input_Registers_In_AT."32085"[13] : Fan volume
   // // Input_Registers_In_AT."32085"[14] : Fan volume
   // // Input_Registers_In_AT."32086"[0] : Operation mode
   // // Input_Registers_In_AT."32086"[1] : Operation mode
   // // Input_Registers_In_AT."32086"[2] : Operation mode
   // // Input_Registers_In_AT."32086"[3] : Operation mode
   // // Input_Registers_In_AT."32086"[4] : Filter sign status
   // // Input_Registers_In_AT."32086"[5] : Filter sign status
   // // Input_Registers_In_AT."32086"[6] : Filter sign status
   // // Input_Registers_In_AT."32086"[7] : Filter sign status
   // // Input_Registers_In_AT."32086"[8] : Operation status
   // // Input_Registers_In_AT."32086"[9] : Operation status
   // // Input_Registers_In_AT."32086"[10] : Operation status
   // // Input_Registers_In_AT."32086"[11] : Operation status
   // // Input_Registers_In_AT."32086"[14] : Cool/Heat Master
   // // Input_Registers_In_AT."32086"[15] : Cool/Heat Master
   // // Input_Registers_In_AT."32087"[15] : Signed Bit
   // // Input_Registers_In_AT."32088"[0] : Error code mapping value1
   // // Input_Registers_In_AT."32088"[1] : Error code mapping value1
   // // Input_Registers_In_AT."32088"[2] : Error code mapping value1
   // // Input_Registers_In_AT."32088"[3] : Error code mapping value1
   // // Input_Registers_In_AT."32088"[4] : Error code mapping value2
   // // Input_Registers_In_AT."32088"[5] : Error code mapping value2
   // // Input_Registers_In_AT."32088"[6] : Error code mapping value2
   // // Input_Registers_In_AT."32088"[7] : Error code mapping value2
   // // Input_Registers_In_AT."32088"[8] : Malfunction
   // // Input_Registers_In_AT."32088"[9] : Warning
   // // Input_Registers_In_AT."32088"[10] : Operation status
   // // Input_Registers_In_AT."32089"[15] : Signed Bit
   // // Input_Registers_In_AT."32090"[8] : Indoor unit temperature sensor error
   // // Input_Registers_In_AT."32090"[15] : Indoor unit temperature sensor data received
   // // Input_Registers_In_AT."32091"[0] : OnOff Status
   // // Input_Registers_In_AT."32091"[2] : Forced off status
   // // Input_Registers_In_AT."32091"[8] : Fan direction
   // // Input_Registers_In_AT."32091"[9] : Fan direction
   // // Input_Registers_In_AT."32091"[10] : Fan direction
   // // Input_Registers_In_AT."32091"[12] : Fan volume
   // // Input_Registers_In_AT."32091"[13] : Fan volume
   // // Input_Registers_In_AT."32091"[14] : Fan volume
   // // Input_Registers_In_AT."32092"[0] : Operation mode
   // // Input_Registers_In_AT."32092"[1] : Operation mode
   // // Input_Registers_In_AT."32092"[2] : Operation mode
   // // Input_Registers_In_AT."32092"[3] : Operation mode
   // // Input_Registers_In_AT."32092"[4] : Filter sign status
   // // Input_Registers_In_AT."32092"[5] : Filter sign status
   // // Input_Registers_In_AT."32092"[6] : Filter sign status
   // // Input_Registers_In_AT."32092"[7] : Filter sign status
   // // Input_Registers_In_AT."32092"[8] : Operation status
   // // Input_Registers_In_AT."32092"[9] : Operation status
   // // Input_Registers_In_AT."32092"[10] : Operation status
   // // Input_Registers_In_AT."32092"[11] : Operation status
   // // Input_Registers_In_AT."32092"[14] : Cool/Heat Master
   // // Input_Registers_In_AT."32092"[15] : Cool/Heat Master
   // // Input_Registers_In_AT."32093"[15] : Signed Bit
   // // Input_Registers_In_AT."32094"[0] : Error code mapping value1
   // // Input_Registers_In_AT."32094"[1] : Error code mapping value1
   // // Input_Registers_In_AT."32094"[2] : Error code mapping value1
   // // Input_Registers_In_AT."32094"[3] : Error code mapping value1
   // // Input_Registers_In_AT."32094"[4] : Error code mapping value2
   // // Input_Registers_In_AT."32094"[5] : Error code mapping value2
   // // Input_Registers_In_AT."32094"[6] : Error code mapping value2
   // // Input_Registers_In_AT."32094"[7] : Error code mapping value2
   // // Input_Registers_In_AT."32094"[8] : Malfunction
   // // Input_Registers_In_AT."32094"[9] : Warning
   // // Input_Registers_In_AT."32094"[10] : Operation status
   // // Input_Registers_In_AT."32095"[15] : Signed Bit
   // // Input_Registers_In_AT."32096"[8] : Indoor unit temperature sensor error
   // // Input_Registers_In_AT."32096"[15] : Indoor unit temperature sensor data received
BEGIN

REGION Network 2: Enable supply voltage diagnostic
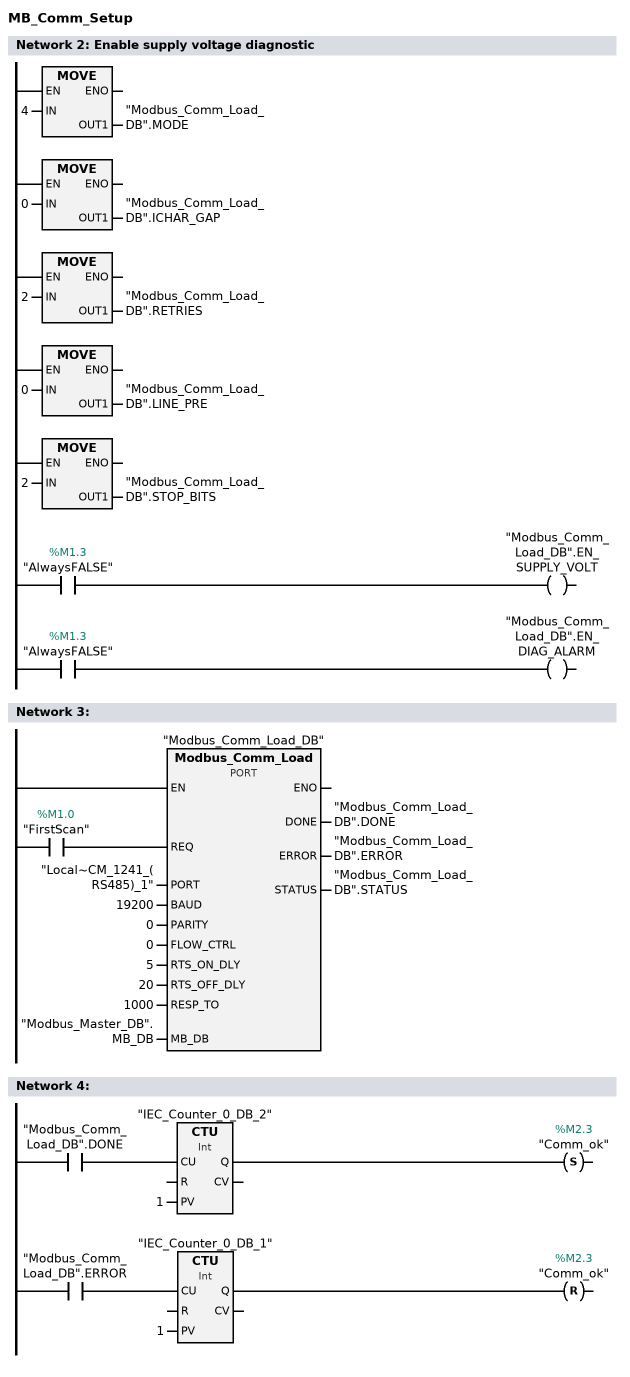
   RUNG wire#powerrail
      Move(in := 4, out1 => "Modbus_Comm_Load_DB".MODE)
   END_RUNG
   RUNG wire#powerrail
      Move(in := 0, out1 => "Modbus_Comm_Load_DB".ICHAR_GAP)
   END_RUNG
   RUNG wire#powerrail
      Move(in := 2, out1 => "Modbus_Comm_Load_DB".RETRIES)
   END_RUNG
   RUNG wire#powerrail
      Move(in := 0, out1 => "Modbus_Comm_Load_DB".LINE_PRE)
   END_RUNG
   RUNG wire#powerrail
      Move(in := 2, out1 => "Modbus_Comm_Load_DB".STOP_BITS)
   END_RUNG
   RUNG wire#powerrail
      Contact( "AlwaysFALSE" )
      Coil( "Modbus_Comm_Load_DB".EN_SUPPLY_VOLT )
   END_RUNG
   RUNG wire#powerrail
      Contact( "AlwaysFALSE" )
      Coil( "Modbus_Comm_Load_DB".EN_DIAG_ALARM )
   END_RUNG
   // the same network as SCL:
   "Modbus_Comm_Load_DB".MODE := 4;
   "Modbus_Comm_Load_DB".ICHAR_GAP := 0;
   "Modbus_Comm_Load_DB".RETRIES := 2;
   "Modbus_Comm_Load_DB".LINE_PRE := 0;
   "Modbus_Comm_Load_DB".STOP_BITS := 2;
   "Modbus_Comm_Load_DB".EN_SUPPLY_VOLT := "AlwaysFALSE";
   "Modbus_Comm_Load_DB".EN_DIAG_ALARM := "AlwaysFALSE";
END_REGION

REGION Network 3
   RUNG wire#powerrail
      { S7_Templates := "[card := 0, port_type := PORT, word_type := UInt, dint_type := UDInt, mbbase_type := P2P_MB_BASE]" } "Modbus_Comm_Load_DB".Modbus_Comm_Load(REQ := wire#w1, PORT := "Local~CM_1241_(RS485)_1", BAUD := 19200, PARITY := 0, FLOW_CTRL := 0, RTS_ON_DLY := 5, RTS_OFF_DLY := 20, RESP_TO := 1000, MB_DB := "Modbus_Master_DB".MB_DB, DONE => "Modbus_Comm_Load_DB".DONE, ERROR => "Modbus_Comm_Load_DB".ERROR, STATUS => "Modbus_Comm_Load_DB".STATUS)
   END_RUNG
   RUNG wire#powerrail
      Contact( "FirstScan" )
   END_RUNG wire#w1
   // the same network as SCL:
   "Modbus_Comm_Load_DB"(REQ := "FirstScan",   // Modbus_Comm_Load
                         PORT := "Local~CM_1241_(RS485)_1",
                         BAUD := 19200,
                         PARITY := 0,
                         FLOW_CTRL := 0,
                         RTS_ON_DLY := 5,
                         RTS_OFF_DLY := 20,
                         RESP_TO := 1000,
                         MB_DB := "Modbus_Master_DB".MB_DB,
                         DONE => "Modbus_Comm_Load_DB".DONE,
                         ERROR => "Modbus_Comm_Load_DB".ERROR,
                         STATUS => "Modbus_Comm_Load_DB".STATUS);
END_REGION

REGION Network 4
   RUNG wire#powerrail
      Contact( "Modbus_Comm_Load_DB".DONE )
      { S7_Templates := "value_type := Int" } "IEC_Counter_0_DB_2".CTU(r :=, pv := 1, cv =>)
      S_Coil( "Comm_ok" )
   END_RUNG
   RUNG wire#powerrail
      Contact( "Modbus_Comm_Load_DB".ERROR )
      { S7_Templates := "value_type := Int" } "IEC_Counter_0_DB_1".CTU(r :=, pv := 1, cv =>)
      R_Coil( "Comm_ok" )
   END_RUNG
   // the same network as SCL:
   "IEC_Counter_0_DB_2".CTU(CU := "Modbus_Comm_Load_DB".DONE, PV := 1);
   IF "IEC_Counter_0_DB_2".Q THEN "Comm_ok" := TRUE; END_IF;
   "IEC_Counter_0_DB_1".CTU(CU := "Modbus_Comm_Load_DB".ERROR, PV := 1);
   IF "IEC_Counter_0_DB_1".Q THEN "Comm_ok" := FALSE; END_IF;
END_REGION
END_FUNCTION_BLOCK

ORGANIZATION_BLOCK "Cyclic interrupt"   // OB30, LAD, CyclicInterrupt
{ S7_Optimized_Access := 'TRUE' }
VERSION : 0.1
// stored: AutoNumber true, IsIECCheckEnabled false, SetENOAutomatically false
   VAR_INPUT
      Initial_Call : Bool;   // Initial call of this OB
      Event_Count : Int;   // Events discarded
   END_VAR
   VAR_TEMP
      Aux_SP_1 : Int;
      Aux_SP_2 : Int;
      Aux_SP_3 : Int;
      Aux_SP_4 : Int;
      Aux_SP_5 : Int;
      Aux_SP_6 : Int;
      Aux_SP_7 : Int;
      Aux_SP_8 : Int;
      Aux_SP_9 : Int;
      Aux_SP_10 : Int;
      Aux_SP_11 : Int;
      Aux_SP_12 : Int;
      Aux_SP_13 : Int;
      Aux_SP_14 : Int;
   END_VAR
   VAR_TEMP   // added for the SCL form of the ladder/FBD networks
      _w1 : Bool;
   END_VAR
BEGIN

REGION Network 2: START
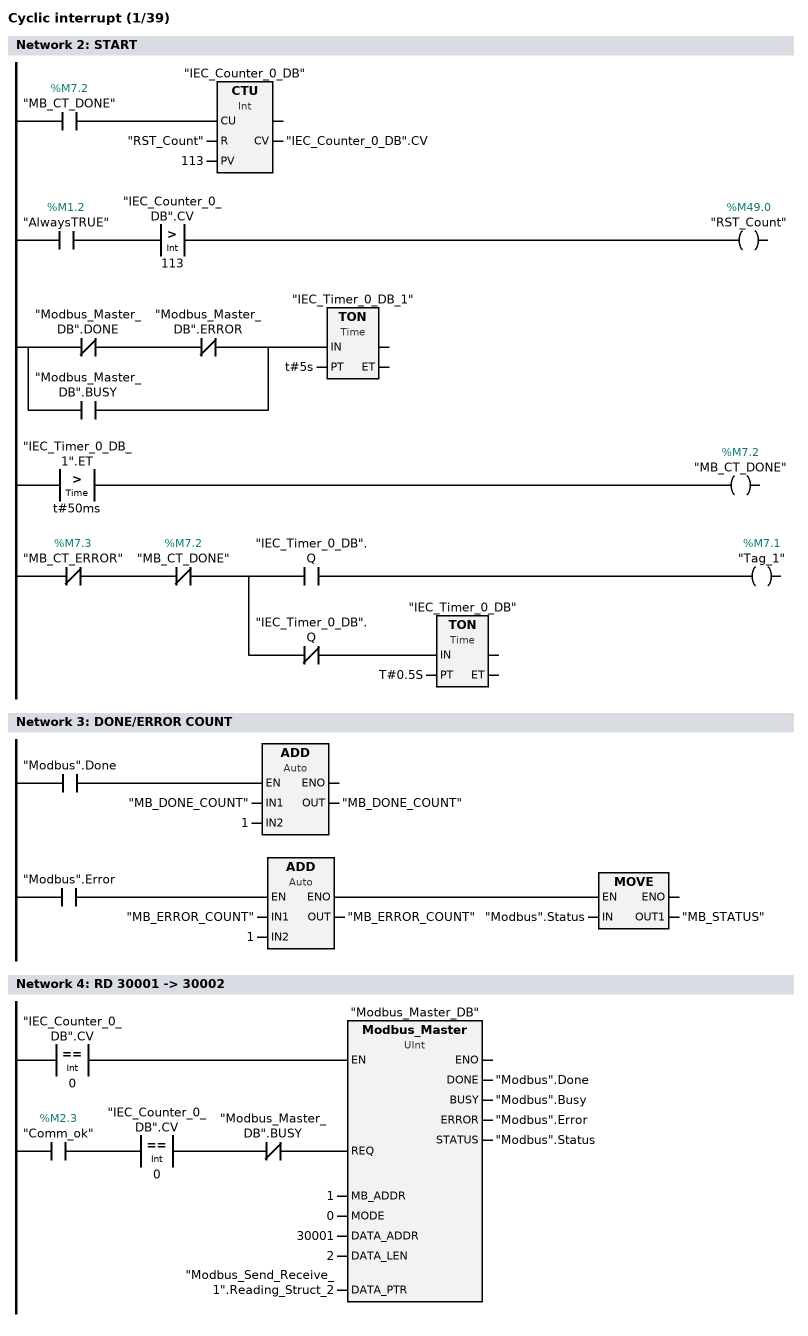
   RUNG wire#powerrail
      Contact( "MB_CT_DONE" )
      { S7_Templates := "value_type := Int" } "IEC_Counter_0_DB".CTU(r := "RST_Count", pv := 113, cv => "IEC_Counter_0_DB".CV)
   END_RUNG
   RUNG wire#powerrail
      Contact( "AlwaysTRUE" )
      { S7_Templates := "SrcType := Int" } GT_Contact(in1 := "IEC_Counter_0_DB".CV, in2 := 113)
      Coil( "RST_Count" )
   END_RUNG
   RUNG wire#powerrail
      I_Contact( "Modbus_Master_DB".DONE )
      I_Contact( "Modbus_Master_DB".ERROR )
      wire#w1
      { S7_Templates := "time_type := Time" } "IEC_Timer_0_DB_1".TON(pt := t#5s, et =>)
   END_RUNG
   RUNG wire#powerrail
      Contact( "Modbus_Master_DB".BUSY )
   END_RUNG wire#w1
   RUNG wire#powerrail
      { S7_Templates := "SrcType := Time" } GT_Contact(in1 := "IEC_Timer_0_DB_1".ET, in2 := t#50ms)
      Coil( "MB_CT_DONE" )
   END_RUNG
   RUNG wire#powerrail
      I_Contact( "MB_CT_ERROR" )
      I_Contact( "MB_CT_DONE" )
      wire#w2
      Contact( "IEC_Timer_0_DB".Q )
      Coil( "Tag_1" )
   END_RUNG
   RUNG wire#w2
      I_Contact( "IEC_Timer_0_DB".Q )
      { S7_Templates := "time_type := Time" } "IEC_Timer_0_DB".TON(pt := T#0.5S, et =>)
   END_RUNG
   // the same network as SCL:
   "IEC_Counter_0_DB".CTU(CU := "MB_CT_DONE", R := "RST_Count", PV := 113, CV => "IEC_Counter_0_DB".CV);
   "RST_Count" := "AlwaysTRUE" AND ("IEC_Counter_0_DB".CV > 113);
   "IEC_Timer_0_DB_1".TON(IN := (NOT "Modbus_Master_DB".DONE AND NOT "Modbus_Master_DB".ERROR) OR "Modbus_Master_DB".BUSY,
                          PT := t#5s);
   "MB_CT_DONE" := "IEC_Timer_0_DB_1".ET > t#50ms;
   #_w1 := NOT "MB_CT_ERROR" AND NOT "MB_CT_DONE";
   "Tag_1" := #_w1 AND "IEC_Timer_0_DB".Q;
   "IEC_Timer_0_DB".TON(IN := #_w1 AND NOT "IEC_Timer_0_DB".Q, PT := T#0.5S);
END_REGION

REGION Network 3: DONE/ERROR COUNT
   RUNG wire#powerrail
      Contact( "Modbus".Done )
      Add(in1 := "MB_DONE_COUNT", in2 := 1, out => "MB_DONE_COUNT")
   END_RUNG
   RUNG wire#powerrail
      Contact( "Modbus".Error )
      Add(in1 := "MB_ERROR_COUNT", in2 := 1, out => "MB_ERROR_COUNT")
      Move(in := "Modbus".Status, out1 => "MB_STATUS")
   END_RUNG
   // the same network as SCL:
   IF "Modbus".Done THEN "MB_DONE_COUNT" := "MB_DONE_COUNT" + 1; END_IF;
   IF "Modbus".Error THEN
       "MB_ERROR_COUNT" := "MB_ERROR_COUNT" + 1;
       "MB_STATUS" := "Modbus".Status;
   END_IF;
END_REGION

REGION Network 4: RD 30001 -> 30002
   RUNG wire#powerrail
      { S7_Templates := "SrcType := Int" } EQ_Contact(in1 := "IEC_Counter_0_DB".CV, in2 := 0)
      { S7_Templates := "[card := 0, word_type := UInt, dword_type := UDInt, byte_type := USInt, any_type := Variant]" } "Modbus_Master_DB".Modbus_Master(REQ := wire#w1, MB_ADDR := 1, MODE := 0, DATA_ADDR := 30001, DATA_LEN := 2, DATA_PTR := "Modbus_Send_Receive_1".Reading_Struct_2, DONE => "Modbus".Done, BUSY => "Modbus".Busy, ERROR => "Modbus".Error, STATUS => "Modbus".Status)
   END_RUNG
   RUNG wire#powerrail
      Contact( "Comm_ok" )
      { S7_Templates := "SrcType := Int" } EQ_Contact(in1 := "IEC_Counter_0_DB".CV, in2 := 0)
      I_Contact( "Modbus_Master_DB".BUSY )
   END_RUNG wire#w1
   // the same network as SCL:
   IF "IEC_Counter_0_DB".CV = 0 THEN
       "Modbus_Master_DB"(REQ := "Comm_ok" AND ("IEC_Counter_0_DB".CV = 0) AND NOT "Modbus_Master_DB".BUSY,   // Modbus_Master
                          MB_ADDR := 1,
                          MODE := 0,
                          DATA_ADDR := 30001,
                          DATA_LEN := 2,
                          DATA_PTR := "Modbus_Send_Receive_1".Reading_Struct_2,
                          DONE => "Modbus".Done,
                          BUSY => "Modbus".Busy,
                          ERROR => "Modbus".Error,
                          STATUS => "Modbus".Status);
   END_IF;
END_REGION

REGION Network 5: STS MAN/AUTO
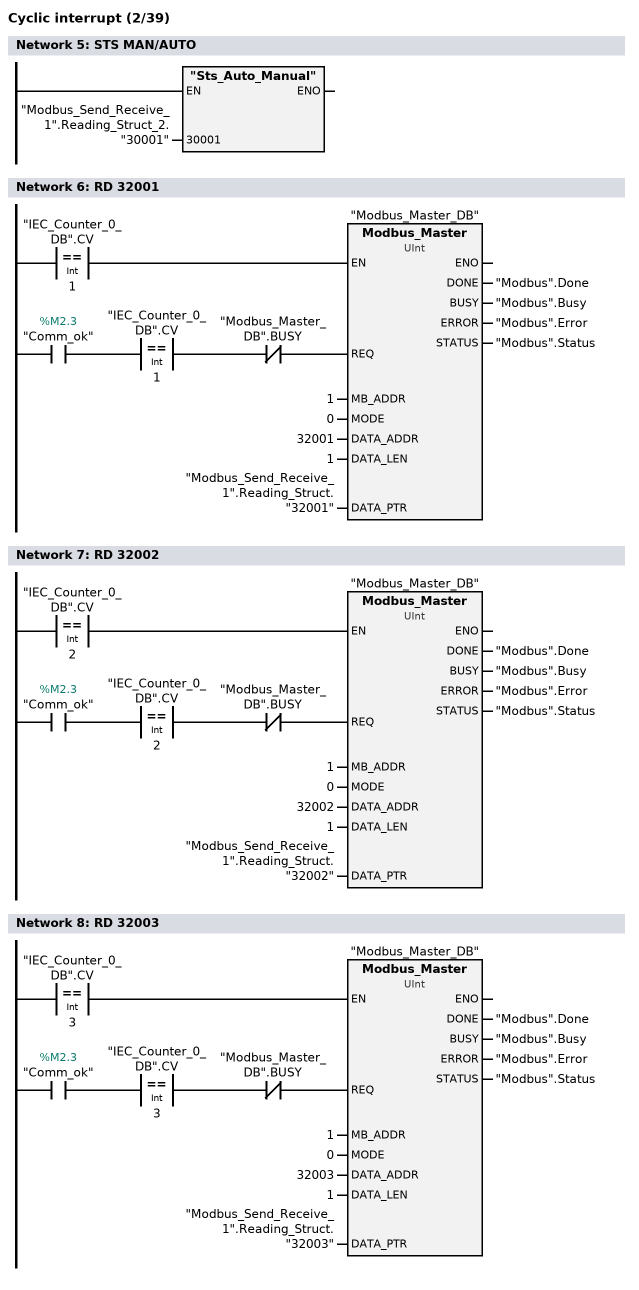
   RUNG wire#powerrail
      "Sts_Auto_Manual"("30001" := "Modbus_Send_Receive_1".Reading_Struct_2."30001")
   END_RUNG
   // the same network as SCL:
   "Sts_Auto_Manual"("30001" := "Modbus_Send_Receive_1".Reading_Struct_2."30001");
END_REGION

REGION Network 6: RD 32001
   RUNG wire#powerrail
      { S7_Templates := "SrcType := Int" } EQ_Contact(in1 := "IEC_Counter_0_DB".CV, in2 := 1)
      { S7_Templates := "[card := 0, word_type := UInt, dword_type := UDInt, byte_type := USInt, any_type := Variant]" } "Modbus_Master_DB".Modbus_Master(REQ := wire#w1, MB_ADDR := 1, MODE := 0, DATA_ADDR := 32001, DATA_LEN := 1, DATA_PTR := "Modbus_Send_Receive_1".Reading_Struct."32001", DONE => "Modbus".Done, BUSY => "Modbus".Busy, ERROR => "Modbus".Error, STATUS => "Modbus".Status)
   END_RUNG
   RUNG wire#powerrail
      Contact( "Comm_ok" )
      { S7_Templates := "SrcType := Int" } EQ_Contact(in1 := "IEC_Counter_0_DB".CV, in2 := 1)
      I_Contact( "Modbus_Master_DB".BUSY )
   END_RUNG wire#w1
   // the same network as SCL:
   IF "IEC_Counter_0_DB".CV = 1 THEN
       "Modbus_Master_DB"(REQ := "Comm_ok" AND ("IEC_Counter_0_DB".CV = 1) AND NOT "Modbus_Master_DB".BUSY,   // Modbus_Master
                          MB_ADDR := 1,
                          MODE := 0,
                          DATA_ADDR := 32001,
                          DATA_LEN := 1,
                          DATA_PTR := "Modbus_Send_Receive_1".Reading_Struct."32001",
                          DONE => "Modbus".Done,
                          BUSY => "Modbus".Busy,
                          ERROR => "Modbus".Error,
                          STATUS => "Modbus".Status);
   END_IF;
END_REGION

